	(*----- EOAT Cable(s) -------*)
	(*Fault901 - EOAT01 Cable(s) disconnected*)
		Fault_Tmrs[901].PT:=No_Timer;
		Fault_Tmrs[901]();
		Fault_Tmrs[901].IN:= (MAIN.R1.FB_In.Options.EOAT_Amount>=1) AND
							((EOAT01.ECatSlave_Cable_Breaks[0]<>0)
								OR (EOAT01.ECatSlave_Cable_Breaks[1]<>0));
		Out_To_ICxx.System_Faults[901]:=Fault_Tmrs[901].Q;
	(*Fault902 - EOAT02 Cable(s) disconnected*)
		Fault_Tmrs[902].PT:=No_Timer;
		Fault_Tmrs[902]();
		Fault_Tmrs[902].IN:= (MAIN.R2.FB_In.Options.EOAT_Amount>=2) AND
							((EOAT02.ECatSlave_Cable_Breaks[0]<>0)
								OR (EOAT02.ECatSlave_Cable_Breaks[1]<>0));
		Out_To_ICxx.System_Faults[902]:=Fault_Tmrs[902].Q;
	(*Fault903 - EOAT03 Cable(s) disconnected*)
		Fault_Tmrs[903].PT:=No_Timer;
		Fault_Tmrs[903]();
		Fault_Tmrs[903].IN:= (MAIN.R3.FB_In.Options.EOAT_Amount>=3) AND
							((EOAT04.ECatSlave_Cable_Breaks[0]<>0)
								OR (EOAT04.ECatSlave_Cable_Breaks[1]<>0));
		Out_To_ICxx.System_Faults[903]:=Fault_Tmrs[903].Q;
	(*Fault904 - EOAT04 Cable(s) disconnected*)
		Fault_Tmrs[904].PT:=No_Timer;
		Fault_Tmrs[904]();
		Fault_Tmrs[904].IN:= (MAIN.R4.FB_In.Options.EOAT_Amount>=4) AND
							((EOAT05.ECatSlave_Cable_Breaks[0]<>0)
								OR (EOAT05.ECatSlave_Cable_Breaks[1]<>0));
		Out_To_ICxx.System_Faults[904]:=Fault_Tmrs[904].Q;
	(*Fault905 - EOAT05 Cable(s) disconnected*)
		Fault_Tmrs[905].PT:=No_Timer;
		Fault_Tmrs[905]();
		Fault_Tmrs[905].IN:= (MAIN.R5.FB_In.Options.EOAT_Amount>=5) AND
							((EOAT05.ECatSlave_Cable_Breaks[0]<>0)
								OR (EOAT05.ECatSlave_Cable_Breaks[1]<>0));
		Out_To_ICxx.System_Faults[905]:=Fault_Tmrs[905].Q;
	(*Fault906 - EOAT06 Cable(s) disconnected*)
		Fault_Tmrs[906].PT:=No_Timer;
		Fault_Tmrs[906]();
		Fault_Tmrs[906].IN:= (MAIN.R6.FB_In.Options.EOAT_Amount>=6) AND
							((EOAT06.ECatSlave_Cable_Breaks[0]<>0)
								OR (EOAT06.ECatSlave_Cable_Breaks[1]<>0));
		Out_To_ICxx.System_Faults[906]:=Fault_Tmrs[906].Q;
	(*Fault907 - EOAT07 Cable(s) disconnected*)
		Fault_Tmrs[907].PT:=No_Timer;
		Fault_Tmrs[907]();
		Fault_Tmrs[907].IN:= (MAIN.R7.FB_In.Options.EOAT_Amount>=7) AND
							((EOAT07.ECatSlave_Cable_Breaks[0]<>0)
								OR (EOAT07.ECatSlave_Cable_Breaks[1]<>0));
		Out_To_ICxx.System_Faults[907]:=Fault_Tmrs[907].Q;
	(*Fault908 - EOAT08 Cable(s) disconnected*)
		Fault_Tmrs[908].PT:=No_Timer;
		Fault_Tmrs[908]();
		Fault_Tmrs[908].IN:= (MAIN.R8.FB_In.Options.EOAT_Amount>=8) AND
							((EOAT08.ECatSlave_Cable_Breaks[0]<>0)
								OR (EOAT08.ECatSlave_Cable_Breaks[1]<>0));
		Out_To_ICxx.System_Faults[908]:=Fault_Tmrs[908].Q;
	(*Fault909 - EOAT09 Cable(s) disconnected*)
		Fault_Tmrs[909].PT:=No_Timer;
		Fault_Tmrs[909]();
		Fault_Tmrs[909].IN:= (MAIN.R9.FB_In.Options.EOAT_Amount>=9) AND
							((EOAT09.ECatSlave_Cable_Breaks[0]<>0)
								OR (EOAT09.ECatSlave_Cable_Breaks[1]<>0));
		Out_To_ICxx.System_Faults[909]:=Fault_Tmrs[909].Q;
	(*Fault910 - EOAT10 Cable(s) disconnected*)
		Fault_Tmrs[820].PT:=No_Timer;
		Fault_Tmrs[820]();
		Fault_Tmrs[820].IN:=(MAIN.R10.FB_In.Options.EOAT_Amount>=10) AND
							((EOAT10.ECatSlave_Cable_Breaks[0]<>0)
								OR (EOAT10.ECatSlave_Cable_Breaks[1]<>0));
		Out_To_ICxx.System_Faults[820]:=Fault_Tmrs[820].Q; 
	(*Fault911 - EOAT11 Cable(s) disconnected*)
		Fault_Tmrs[911].PT:=No_Timer;
		Fault_Tmrs[911]();
		Fault_Tmrs[911].IN:= FALSE;
		Out_To_ICxx.System_Faults[911]:=Fault_Tmrs[911].Q;
	(*Fault912 - EOAT12 Cable(s) disconnected*)
		Fault_Tmrs[912].PT:=No_Timer;
		Fault_Tmrs[912]();
		Fault_Tmrs[912].IN:= FALSE;
		Out_To_ICxx.System_Faults[912]:=Fault_Tmrs[912].Q;
	(*Fault913 - EOAT13 Cable(s) disconnected*)
		Fault_Tmrs[913].PT:=No_Timer;
		Fault_Tmrs[913]();
		Fault_Tmrs[913].IN:= FALSE;
		Out_To_ICxx.System_Faults[913]:=Fault_Tmrs[913].Q;
	(*Fault914 - EOAT14 Cable(s) disconnected*)
		Fault_Tmrs[914].PT:=No_Timer;
		Fault_Tmrs[914]();
		Fault_Tmrs[914].IN:= FALSE;
		Out_To_ICxx.System_Faults[914]:=Fault_Tmrs[914].Q;
	(*Fault915 - EOAT15 Cable(s) disconnected*)
		Fault_Tmrs[915].PT:=No_Timer;
		Fault_Tmrs[915]();
		Fault_Tmrs[915].IN:= FALSE;
		Out_To_ICxx.System_Faults[915]:=Fault_Tmrs[915].Q;
	(*Fault916 - EOAT16 Cable(s) disconnected*)
		Fault_Tmrs[916].PT:=No_Timer;
		Fault_Tmrs[916]();
		Fault_Tmrs[916].IN:= FALSE;
		Out_To_ICxx.System_Faults[916]:=Fault_Tmrs[916].Q;
	(*Fault917 - EOAT17 Cable(s) disconnected*)
		Fault_Tmrs[917].PT:=No_Timer;
		Fault_Tmrs[917]();
		Fault_Tmrs[917].IN:= FALSE;
		Out_To_ICxx.System_Faults[917]:=Fault_Tmrs[917].Q;
	(*Fault918 - EOAT18 Cable(s) disconnected*)
		Fault_Tmrs[918].PT:=No_Timer;
		Fault_Tmrs[918]();
		Fault_Tmrs[918].IN:= FALSE;
		Out_To_ICxx.System_Faults[918]:=Fault_Tmrs[918].Q;
	(*Fault919 - EOAT19 Cable(s) disconnected*)
		Fault_Tmrs[919].PT:=No_Timer;
		Fault_Tmrs[919]();
		Fault_Tmrs[919].IN:= FALSE;
		Out_To_ICxx.System_Faults[919]:=Fault_Tmrs[919].Q;
	(*Fault920 - EOAT20 Cable(s) disconnected*)
		Fault_Tmrs[920].PT:=No_Timer;
		Fault_Tmrs[920]();
		Fault_Tmrs[920].IN:= FALSE;
		Out_To_ICxx.System_Faults[920]:=Fault_Tmrs[920].Q;
	(*Fault921 - EOAT21 Cable(s) disconnected*)
		Fault_Tmrs[921].PT:=No_Timer;
		Fault_Tmrs[921]();
		Fault_Tmrs[921].IN:= FALSE;
		Out_To_ICxx.System_Faults[921]:=Fault_Tmrs[921].Q;
	(*Fault922 - EOAT22 Cable(s) disconnected*)
		Fault_Tmrs[922].PT:=No_Timer;
		Fault_Tmrs[922]();
		Fault_Tmrs[922].IN:= FALSE;
		Out_To_ICxx.System_Faults[922]:=Fault_Tmrs[922].Q;
	(*Fault923 - EOAT23 Cable(s) disconnected*)
		Fault_Tmrs[923].PT:=No_Timer;
		Fault_Tmrs[923]();
		Fault_Tmrs[923].IN:= FALSE;
		Out_To_ICxx.System_Faults[923]:=Fault_Tmrs[923].Q;
	(*Fault924 - EOAT24 Cable(s) disconnected*)
		Fault_Tmrs[924].PT:=No_Timer;
		Fault_Tmrs[924]();
		Fault_Tmrs[924].IN:= FALSE;
		Out_To_ICxx.System_Faults[924]:=Fault_Tmrs[924].Q;
	(*Fault925 - EOAT25 Cable(s) disconnected*)
		Fault_Tmrs[925].PT:=No_Timer;
		Fault_Tmrs[925]();
		Fault_Tmrs[925].IN:= FALSE;
		Out_To_ICxx.System_Faults[925]:=Fault_Tmrs[925].Q;
	(*Fault926 - EOAT26 Cable(s) disconnected*)
		Fault_Tmrs[926].PT:=No_Timer;
		Fault_Tmrs[926]();
		Fault_Tmrs[926].IN:= FALSE;
		Out_To_ICxx.System_Faults[926]:=Fault_Tmrs[926].Q;
	(*Fault927 - EOAT27 Cable(s) disconnected*)
		Fault_Tmrs[927].PT:=No_Timer;
		Fault_Tmrs[927]();
		Fault_Tmrs[927].IN:= FALSE;
		Out_To_ICxx.System_Faults[927]:=Fault_Tmrs[927].Q;
	(*Fault928 - EOAT28 Cable(s) disconnected*)
		Fault_Tmrs[928].PT:=No_Timer;
		Fault_Tmrs[928]();
		Fault_Tmrs[928].IN:= FALSE;
		Out_To_ICxx.System_Faults[928]:=Fault_Tmrs[928].Q;
	(*Fault929 - EOAT29 Cable(s) disconnected*)
		Fault_Tmrs[929].PT:=No_Timer;
		Fault_Tmrs[929]();
		Fault_Tmrs[929].IN:= FALSE;
		Out_To_ICxx.System_Faults[929]:=Fault_Tmrs[929].Q;
	(*Fault930 - EOAT30 Cable(s) disconnected*)
		Fault_Tmrs[930].PT:=No_Timer;
		Fault_Tmrs[930]();
		Fault_Tmrs[930].IN:= FALSE;
		Out_To_ICxx.System_Faults[930]:=Fault_Tmrs[930].Q;


	(* --------------------------Services Stand Cable Faults----------------------------*)
	(*Fault931 - SS01 IN Cable Fault*)
		Fault_Tmrs[931].PT:=No_Timer;
		Fault_Tmrs[931]();
		Fault_Tmrs[931].IN:= GTAC_CONFIG.Option_Air1  AND
							MAIN.SS01.EP2028_NotPresent;
		Out_To_ICxx.System_Faults[931]:=Fault_Tmrs[931].Q;
	(*Fault932 - SS01 OUT Cable Fault*)
		Fault_Tmrs[932].PT:=No_Timer;
		Fault_Tmrs[932]();
		Fault_Tmrs[932].IN:= GTAC_CONFIG.Option_Air1  AND
							MAIN.SS01.EP1008_PortB_MissingLink;
		Out_To_ICxx.System_Faults[932]:=Fault_Tmrs[932].Q;
	(*Fault933 - SS02 IN Cable Fault*)
		Fault_Tmrs[933].PT:=No_Timer;
		Fault_Tmrs[933]();
		Fault_Tmrs[933].IN:= GTAC_CONFIG.Option_Air2  AND
							MAIN.SS02.EP2028_NotPresent;
		Out_To_ICxx.System_Faults[933]:=Fault_Tmrs[933].Q;
	(*Fault934 - SS02 OUT Cable Fault*)
		Fault_Tmrs[934].PT:=No_Timer;
		Fault_Tmrs[934]();
		Fault_Tmrs[934].IN:= GTAC_CONFIG.Option_Air2  AND
							MAIN.SS02.EP1008_PortB_MissingLink;
		Out_To_ICxx.System_Faults[934]:=Fault_Tmrs[934].Q;
(*
	(*Fault935 - SS03 IN Cable Fault*)
		Fault_Tmrs[935].PT:=No_Timer;
		Fault_Tmrs[935]();
		Fault_Tmrs[935].IN:= (GTAC_CONFIG.Option_Air1>=1)  AND
							MAIN.SS03.EP2028_NotPresent;
		Out_To_ICxx.System_Faults[935]:=Fault_Tmrs[935].Q;
	(*Fault936 - SS03 OUT Cable Fault*)
		Fault_Tmrs[936].PT:=No_Timer;
		Fault_Tmrs[936]();
		Fault_Tmrs[936].IN:= (GTAC_CONFIG.Option_Air1>=1)  AND
							MAIN.SS03.EP1008_PortB_MissingLink;
		Out_To_ICxx.System_Faults[936]:=Fault_Tmrs[546].Q;
*)
	(* --------------------------Enable Switch Plate Cable Faults----------------------------*)
	(*Fault937 - ESW01 IN Cable Fault*)
		Fault_Tmrs[937].PT:=No_Timer;
		Fault_Tmrs[937]();
		Fault_Tmrs[937].IN:= (GTAC_CONFIG.Option_ESW_Count>=1)  AND
							MAIN.ESW01.EP1908_NotPresent;
		Out_To_ICxx.System_Faults[937]:=Fault_Tmrs[937].Q;
	(*Fault938 - ESW01 OUT Cable Fault*)
		Fault_Tmrs[938].PT:=No_Timer;
		Fault_Tmrs[938]();
		Fault_Tmrs[938].IN:= (GTAC_CONFIG.Option_ESW_Count>=1)  AND
							MAIN.ESW01.EP1908_PortB_MissingLink;
		Out_To_ICxx.System_Faults[938]:=Fault_Tmrs[938].Q;
	(*Fault939 - ESW02 IN Cable Fault*)
		Fault_Tmrs[939].PT:=No_Timer;
		Fault_Tmrs[939]();
		Fault_Tmrs[939].IN:= (GTAC_CONFIG.Option_ESW_Count>=2)  AND
							MAIN.ESW02.EP1908_NotPresent;
		Out_To_ICxx.System_Faults[939]:=Fault_Tmrs[939].Q;
	(*Fault940 - ESW02 OUT Cable Fault*)
		Fault_Tmrs[940].PT:=No_Timer;
		Fault_Tmrs[940]();
		Fault_Tmrs[940].IN:= (GTAC_CONFIG.Option_ESW_Count>=2)  AND
							MAIN.ESW02.EP1908_PortB_MissingLink;
		Out_To_ICxx.System_Faults[940]:=Fault_Tmrs[940].Q;
	(*Fault941 - ESW03 IN Cable Fault*)
		Fault_Tmrs[941].PT:=No_Timer;
		Fault_Tmrs[941]();
		Fault_Tmrs[941].IN:= (GTAC_CONFIG.Option_ESW_Count>=3)  AND
							MAIN.ESW03.EP1908_NotPresent;
		Out_To_ICxx.System_Faults[941]:=Fault_Tmrs[941].Q;
	(*Fault942 - ESW03 OUT Cable Fault*)
		Fault_Tmrs[942].PT:=No_Timer;
		Fault_Tmrs[942]();
		Fault_Tmrs[942].IN:= (GTAC_CONFIG.Option_ESW_Count>=3)  AND
							MAIN.ESW03.EP1908_PortB_MissingLink;
		Out_To_ICxx.System_Faults[942]:=Fault_Tmrs[942].Q;
	(*Fault943 - ESW04 IN Cable Fault*)
		Fault_Tmrs[943].PT:=No_Timer;
		Fault_Tmrs[943]();
		Fault_Tmrs[943].IN:= (GTAC_CONFIG.Option_ESW_Count>=4)  AND
							MAIN.ESW04.EP1908_NotPresent;
		Out_To_ICxx.System_Faults[943]:=Fault_Tmrs[943].Q;
	(*Fault944 - ESW04 OUT Cable Fault*)
		Fault_Tmrs[944].PT:=No_Timer;
		Fault_Tmrs[944]();
		Fault_Tmrs[944].IN:= (GTAC_CONFIG.Option_ESW_Count>=4)  AND
							MAIN.ESW04.EP1908_PortB_MissingLink;
		Out_To_ICxx.System_Faults[944]:=Fault_Tmrs[944].Q;

(* -------------------------- IS Cable Faults----------------------------*)

	(*Fault751 - IS01 Cable break fault (any cable break)*)
		Fault_Tmrs[945].PT:= No_Timer;
		Fault_Tmrs[945]();
		Fault_Tmrs[945].IN:= (GTAC_CONFIG.Option_IS_Count >= 1) AND 
							(MAIN.IS01.ECatSlave_Cable_Breaks <> 0);
		Out_To_ICxx.System_Faults[945]:=Fault_Tmrs[945].Q;
	(*Fault752 - IS01 Profibus Network Fault*)
		Fault_Tmrs[946].PT:= No_Timer;
		Fault_Tmrs[946]();
		Fault_Tmrs[946].IN:= (GTAC_CONFIG.Option_IS_Count >= 1) AND 
							MAIN.IS01.FB_In.Option_Enable_Pbus AND
							NOT (MAIN.IS01.ProfiNode_OK);
		Out_To_ICxx.System_Faults[946]:=Fault_Tmrs[946].Q;

	(* -------------------------- Servo Drive Cable Faults----------------------------*)

	(*Fault951 - SD1 Cable(s) disconnected*)
		Fault_Tmrs[951].PT:= No_Timer;
		Fault_Tmrs[951]();
		Fault_Tmrs[951].IN:= (GTAC_CONFIG.Option_SD_Count>=1) AND
							(Servo_Motion.SD[1].ECatSlave_Cable_Breaks<>0);
		Out_To_ICxx.System_Faults[951]:=Fault_Tmrs[951].Q;
	(*Fault952 - SD2 Cable(s) disconnected*)
		Fault_Tmrs[952].PT:= No_Timer;
		Fault_Tmrs[952]();
		Fault_Tmrs[952].IN:= (GTAC_CONFIG.Option_SD_Count>=2) AND
							(Servo_Motion.SD[2].ECatSlave_Cable_Breaks<>0);
		Out_To_ICxx.System_Faults[952]:=Fault_Tmrs[952].Q;
	(*Fault953 - SD3 Cable(s) disconnected*)
		Fault_Tmrs[953].PT:= No_Timer;
		Fault_Tmrs[953]();
		Fault_Tmrs[953].IN:= (GTAC_CONFIG.Option_SD_Count>=3) AND
							(Servo_Motion.SD[3].ECatSlave_Cable_Breaks<>0);
		Out_To_ICxx.System_Faults[953]:=Fault_Tmrs[953].Q;
	(*Fault954 - SD4 Cable(s) disconnected*)
		Fault_Tmrs[954].PT:= No_Timer;
		Fault_Tmrs[954]();
		Fault_Tmrs[954].IN:= (GTAC_CONFIG.Option_SD_Count>=4) AND
							(Servo_Motion.SD[4].ECatSlave_Cable_Breaks<>0);
		Out_To_ICxx.System_Faults[954]:=Fault_Tmrs[954].Q;
	(*Fault955 - SD5 Cable(s) disconnected*)
		Fault_Tmrs[955].PT:= No_Timer;
		Fault_Tmrs[955]();
		Fault_Tmrs[955].IN:= (GTAC_CONFIG.Option_SD_Count>=5) AND
							(Servo_Motion.SD[5].ECatSlave_Cable_Breaks<>0);
		Out_To_ICxx.System_Faults[955]:=Fault_Tmrs[955].Q;
	(*Fault956 - SD6 Cable(s) disconnected*)
		Fault_Tmrs[956].PT:= No_Timer;
		Fault_Tmrs[956]();
		Fault_Tmrs[956].IN:= (GTAC_CONFIG.Option_SD_Count>=6) AND
							(Servo_Motion.SD[6].ECatSlave_Cable_Breaks<>0);
		Out_To_ICxx.System_Faults[956]:=Fault_Tmrs[956].Q;
	(*Fault957 - SD7 Cable(s) disconnected*)
		Fault_Tmrs[957].PT:= No_Timer;
		Fault_Tmrs[957]();
		Fault_Tmrs[957].IN:= (GTAC_CONFIG.Option_SD_Count>=7) AND
							(Servo_Motion.SD[7].ECatSlave_Cable_Breaks<>0);
		Out_To_ICxx.System_Faults[957]:=Fault_Tmrs[957].Q;
	(*Fault958 - SD8 Cable(s) disconnected*)
		Fault_Tmrs[958].PT:= No_Timer;
		Fault_Tmrs[958]();
		Fault_Tmrs[958].IN:= (GTAC_CONFIG.Option_SD_Count>=8) AND
							(Servo_Motion.SD[8].ECatSlave_Cable_Breaks<>0);
		Out_To_ICxx.System_Faults[958]:=Fault_Tmrs[958].Q;
	(*Fault959 - SD9 Cable(s) disconnected*)
		Fault_Tmrs[959].PT:= No_Timer;
		Fault_Tmrs[959]();
		Fault_Tmrs[959].IN:= (GTAC_CONFIG.Option_SD_Count>=9) AND
							(Servo_Motion.SD[9].ECatSlave_Cable_Breaks<>0);
		Out_To_ICxx.System_Faults[959]:=Fault_Tmrs[959].Q;
	(*Fault960 - SD10 Cable(s) disconnected*)
		Fault_Tmrs[960].PT:= No_Timer;
		Fault_Tmrs[960]();
		Fault_Tmrs[960].IN:= (GTAC_CONFIG.Option_SD_Count>=10) AND
							(Servo_Motion.SD[10].ECatSlave_Cable_Breaks<>0);
		Out_To_ICxx.System_Faults[960]:=Fault_Tmrs[960].Q;
	(*Fault961 - SD11 Cable(s) disconnected*)
		Fault_Tmrs[961].PT:= No_Timer;
		Fault_Tmrs[961]();
		Fault_Tmrs[961].IN:= (GTAC_CONFIG.Option_SD_Count>=11) AND
							(Servo_Motion.SD[11].ECatSlave_Cable_Breaks<>0);
		Out_To_ICxx.System_Faults[961]:=Fault_Tmrs[961].Q;
	(*Fault962 - SD12 Cable(s) disconnected*)
		Fault_Tmrs[962].PT:= No_Timer;
		Fault_Tmrs[962]();
		Fault_Tmrs[962].IN:= (GTAC_CONFIG.Option_SD_Count>=12) AND
							(Servo_Motion.SD[12].ECatSlave_Cable_Breaks<>0);
		Out_To_ICxx.System_Faults[962]:=Fault_Tmrs[962].Q;
	(*Fault963 - SD13 Cable(s) disconnected*)
		Fault_Tmrs[963].PT:= No_Timer;
		Fault_Tmrs[963]();
		Fault_Tmrs[963].IN:= (GTAC_CONFIG.Option_SD_Count>=13) AND
							(Servo_Motion.SD[13].ECatSlave_Cable_Breaks<>0);
		Out_To_ICxx.System_Faults[963]:=Fault_Tmrs[963].Q;
	(*Fault964 - SD14 Cable(s) disconnected*)
		Fault_Tmrs[964].PT:= No_Timer;
		Fault_Tmrs[964]();
		Fault_Tmrs[964].IN:= (GTAC_CONFIG.Option_SD_Count>=14) AND
							(Servo_Motion.SD[14].ECatSlave_Cable_Breaks<>0);
		Out_To_ICxx.System_Faults[964]:=Fault_Tmrs[964].Q;
	(*Fault965 - SD15 Cable(s) disconnected*)
		Fault_Tmrs[965].PT:= No_Timer;
		Fault_Tmrs[965]();
		Fault_Tmrs[965].IN:= (GTAC_CONFIG.Option_SD_Count>=15) AND
							(Servo_Motion.SD[15].ECatSlave_Cable_Breaks<>0);
		Out_To_ICxx.System_Faults[965]:=Fault_Tmrs[965].Q;
	(*Fault966 - SD16 Cable(s) disconnected*)
		Fault_Tmrs[966].PT:= No_Timer;
		Fault_Tmrs[966]();
		Fault_Tmrs[966].IN:= (GTAC_CONFIG.Option_SD_Count>=16) AND
							(Servo_Motion.SD[16].ECatSlave_Cable_Breaks<>0);
		Out_To_ICxx.System_Faults[966]:=Fault_Tmrs[966].Q;
	(*Fault967 - SD17 Cable(s) disconnected*)
		Fault_Tmrs[967].PT:= No_Timer;
		Fault_Tmrs[967]();
		Fault_Tmrs[967].IN:= (GTAC_CONFIG.Option_SD_Count>=17) AND
							(Servo_Motion.SD[17].ECatSlave_Cable_Breaks<>0);
		Out_To_ICxx.System_Faults[967]:=Fault_Tmrs[967].Q;
	(*Fault968 - SD18 Cable(s) disconnected*)
		Fault_Tmrs[968].PT:= No_Timer;
		Fault_Tmrs[968]();
		Fault_Tmrs[968].IN:= (GTAC_CONFIG.Option_SD_Count>=18) AND
							(Servo_Motion.SD[18].ECatSlave_Cable_Breaks<>0);
		Out_To_ICxx.System_Faults[968]:=Fault_Tmrs[968].Q;
	(*Fault969 - SD19 Cable(s) disconnected*)
		Fault_Tmrs[969].PT:= No_Timer;
		Fault_Tmrs[969]();
		Fault_Tmrs[969].IN:= (GTAC_CONFIG.Option_SD_Count>=19) AND
							(Servo_Motion.SD[19].ECatSlave_Cable_Breaks<>0);
		Out_To_ICxx.System_Faults[969]:=Fault_Tmrs[969].Q;
	(*Fault970 - SD20 Cable(s) disconnected*)
		Fault_Tmrs[970].PT:= No_Timer;
		Fault_Tmrs[970]();
		Fault_Tmrs[970].IN:= (GTAC_CONFIG.Option_SD_Count>=20) AND
							(Servo_Motion.SD[20].ECatSlave_Cable_Breaks<>0);
		Out_To_ICxx.System_Faults[970]:=Fault_Tmrs[970].Q;
	(*Fault971 - SD21 Cable(s) disconnected*)
		Fault_Tmrs[971].PT:= No_Timer;
		Fault_Tmrs[971]();
		Fault_Tmrs[971].IN:= (GTAC_CONFIG.Option_SD_Count>=21) AND
							(Servo_Motion.SD[21].ECatSlave_Cable_Breaks<>0);
		Out_To_ICxx.System_Faults[971]:=Fault_Tmrs[971].Q;
	(*Fault972 - SD22 Cable(s) disconnected*)
		Fault_Tmrs[972].PT:= No_Timer;
		Fault_Tmrs[972]();
		Fault_Tmrs[972].IN:= (GTAC_CONFIG.Option_SD_Count>=22) AND
							(Servo_Motion.SD[22].ECatSlave_Cable_Breaks<>0);
		Out_To_ICxx.System_Faults[972]:=Fault_Tmrs[972].Q;
	(*Fault973 - SD23 Cable(s) disconnected*)
		Fault_Tmrs[973].PT:= No_Timer;
		Fault_Tmrs[973]();
		Fault_Tmrs[973].IN:= (GTAC_CONFIG.Option_SD_Count>=23) AND
							(Servo_Motion.SD[23].ECatSlave_Cable_Breaks<>0);
		Out_To_ICxx.System_Faults[973]:=Fault_Tmrs[973].Q;
	(*Fault974 - SD24 Cable(s) disconnected*)
		Fault_Tmrs[974].PT:= No_Timer;
		Fault_Tmrs[974]();
		Fault_Tmrs[974].IN:= (GTAC_CONFIG.Option_SD_Count>=24) AND
							(Servo_Motion.SD[24].ECatSlave_Cable_Breaks<>0);
		Out_To_ICxx.System_Faults[974]:=Fault_Tmrs[974].Q;
	(*Fault975 - SD25 Cable(s) disconnected*)
		Fault_Tmrs[975].PT:= No_Timer;
		Fault_Tmrs[975]();
		Fault_Tmrs[975].IN:= (GTAC_CONFIG.Option_SD_Count>=25) AND
							(Servo_Motion.SD[25].ECatSlave_Cable_Breaks<>0);
		Out_To_ICxx.System_Faults[975]:=Fault_Tmrs[975].Q;
	(*Fault976 - SD26 Cable(s) disconnected*)
		Fault_Tmrs[976].PT:= No_Timer;
		Fault_Tmrs[976]();
		Fault_Tmrs[976].IN:= (GTAC_CONFIG.Option_SD_Count>=26) AND
							(Servo_Motion.SD[26].ECatSlave_Cable_Breaks<>0);
		Out_To_ICxx.System_Faults[976]:=Fault_Tmrs[976].Q;
	(*Fault977 - SD27 Cable(s) disconnected*)
		Fault_Tmrs[977].PT:= No_Timer;
		Fault_Tmrs[977]();
		Fault_Tmrs[977].IN:= (GTAC_CONFIG.Option_SD_Count>=27) AND
							(Servo_Motion.SD[27].ECatSlave_Cable_Breaks<>0);
		Out_To_ICxx.System_Faults[977]:=Fault_Tmrs[977].Q;
	(*Fault978 - SD28 Cable(s) disconnected*)
		Fault_Tmrs[978].PT:= No_Timer;
		Fault_Tmrs[978]();
		Fault_Tmrs[978].IN:= (GTAC_CONFIG.Option_SD_Count>=28) AND
							(Servo_Motion.SD[28].ECatSlave_Cable_Breaks<>0);
		Out_To_ICxx.System_Faults[978]:=Fault_Tmrs[978].Q;
	(*Fault979 - SD29 Cable(s) disconnected*)
		Fault_Tmrs[979].PT:= No_Timer;
		Fault_Tmrs[979]();
		Fault_Tmrs[979].IN:= (GTAC_CONFIG.Option_SD_Count>=29) AND
							(Servo_Motion.SD[29].ECatSlave_Cable_Breaks<>0);
		Out_To_ICxx.System_Faults[979]:=Fault_Tmrs[979].Q;
	(*Fault980 - SD30 Cable(s) disconnected*)
		Fault_Tmrs[980].PT:= No_Timer;
		Fault_Tmrs[980]();
		Fault_Tmrs[980].IN:= (GTAC_CONFIG.Option_SD_Count>=30) AND
							(Servo_Motion.SD[30].ECatSlave_Cable_Breaks<>0);
		Out_To_ICxx.System_Faults[980]:=Fault_Tmrs[980].Q;


	(* --------------------------Laser Controller Cable Faults----------------------------*)
	(*Fault981 - LSR01 IN Cable Fault*)
		Fault_Tmrs[981].PT:=No_Timer;
		Fault_Tmrs[981]();
		Fault_Tmrs[981].IN:= (GTAC_CONFIG.Option_LaserController_Count>=1)  AND
							MAIN.Laser01.EL6692_NotPresent;
		Out_To_ICxx.System_Faults[981]:=Fault_Tmrs[981].Q;
	(*Fault982 - LSR01 OUT Cable Fault*)
		Fault_Tmrs[982].PT:=No_Timer;
		Fault_Tmrs[982]();
		Fault_Tmrs[982].IN:= (GTAC_CONFIG.Option_LaserController_Count>=1)  AND
							MAIN.Laser01.EL6692_PortC_MissingLink;
		Out_To_ICxx.System_Faults[982]:=Fault_Tmrs[982].Q;

	(*------------------------------------------------------------- Start Of Faults that Will NOT Stop All Automation --------------------------------------------------*)
	(*--------------------------------------------------------- Start of  ICxx Operator Station Faults ---------------------------------------------------------*)
	(*------------------- IC01 -----------------*)
	(*Fault991 - IC01OP1 Motion Faults*)
		Fault_Tmrs[991].PT:=Short_Faults;
		Fault_Tmrs[991]();
		Fault_Tmrs[991].IN:= GTAC_CONFIG.Option_HumanFix_Enables.1 AND
							Out_To_ICxx.Fix01_Discrete_Image.CLFaulted.0;
		Out_To_ICxx.System_Faults[991]:=Fault_Tmrs[991].Q;
	(*Fault992 - IC01OP1 Part Present Faults*)
		Fault_Tmrs[992].PT:=Short_Faults;
		Fault_Tmrs[992]();
		Fault_Tmrs[992].IN:= GTAC_CONFIG.Option_HumanFix_Enables.1 AND
							Out_To_ICxx.Fix01_Discrete_Image.PPFaulted.0;
		Out_To_ICxx.System_Faults[992]:=Fault_Tmrs[992].Q;
	(*Fault993 - IC01OP1 Vertical LC Broken While Robot(s) In Zone*)
		VLC_Capture11_TOF.PT:= T#2.0S;
		VLC_Capture11_TOF();
		(*Differentiate between Turtable type Fix01/02 and standard Fix01*)
		(*Turntable Type*)
		IF (MAIN.R1.FB_In.Robot_Type = KUKA_KRC4_SAFEOP_TurnTable) THEN
		VLC_Capture11_TOF.IN:= (GTAC_CONFIG.Option_IC_Count>=1) AND GTAC_CONFIG.Option_HumanFix_Enables.1 AND
								NOT MAIN.IC01.OP1_HumanVertLC_Clear AND NOT Fix01.All_Robots_Clear
								AND (Fix01.Turntable_WorkingOK OR Fix02.Turntable_WorkingOK);
		(*Standard Type*)						
		ELSE
		VLC_Capture11_TOF.IN:= (GTAC_CONFIG.Option_IC_Count>=1) AND GTAC_CONFIG.Option_HumanFix_Enables.1 AND
								NOT MAIN.IC01.OP1_HumanVertLC_Clear AND NOT Fix01.All_Robots_Clear;
		END_IF
		Out_To_ICxx.System_Faults[993]:= VLC_Capture11_TOF.Q;
	(*Fault994 - IC01OP1 Horizontal LC Broken While Robot(s) In Zone*)
		HLC_Capture12_TOF.PT:= T#2.0S;
		HLC_Capture12_TOF();
		(*Differentiate between Turtable type Fix01/02 and standard Fix01*)
		(*Turntable Type*)
		IF (MAIN.R1.FB_In.Robot_Type = KUKA_KRC4_SAFEOP_TurnTable) THEN
		HLC_Capture12_TOF.IN:= (GTAC_CONFIG.Option_IC_Count>=1) AND GTAC_CONFIG.Option_HumanFix_Enables.1 AND
								NOT MAIN.IC01.OP1_HumanHorizLC_Clear AND NOT Fix01.All_Robots_Clear
								AND (Fix01.Turntable_WorkingOK OR Fix02.Turntable_WorkingOK);
		(*Standard Type*)						
		ELSE
		HLC_Capture12_TOF.IN:= (GTAC_CONFIG.Option_IC_Count>=1) AND GTAC_CONFIG.Option_HumanFix_Enables.1 AND
								NOT MAIN.IC01.OP1_HumanHorizLC_Clear AND NOT Fix01.All_Robots_Clear;
		END_IF
		Out_To_ICxx.System_Faults[994]:= HLC_Capture12_TOF.Q;
	(*Fault995 - IC01OP1 Horizontal LC3 Broken While Robot(s) In Zone*)
		HLC_Capture13_TOF.PT:= T#2.0S;
		HLC_Capture13_TOF();
		(*Differentiate between Turtable type Fix01/02 and standard Fix01*)
		(*Turntable Type*)
		IF (MAIN.R1.FB_In.Robot_Type = KUKA_KRC4_SAFEOP_TurnTable) THEN
		HLC_Capture13_TOF.IN:= (GTAC_CONFIG.Option_IC_Count>=1) AND GTAC_CONFIG.Option_HumanFix_Enables.1 AND
								NOT MAIN.IC01.OP1_RobotVertLC_Clear AND NOT Fix01.All_Robots_Clear
								AND (Fix01.Turntable_WorkingOK OR Fix02.Turntable_WorkingOK);
		(*Standard Type*)						
		ELSE
		HLC_Capture13_TOF.IN:= (GTAC_CONFIG.Option_IC_Count>=1) AND GTAC_CONFIG.Option_HumanFix_Enables.1 AND
								NOT MAIN.IC01.OP1_RobotVertLC_Clear AND NOT Fix01.All_Robots_Clear;
		END_IF
		Out_To_ICxx.System_Faults[995]:= HLC_Capture13_TOF.Q;

	(*Fault996 - IC01OP2 Motion Faults*)
		Fault_Tmrs[996].PT:=Short_Faults;
		Fault_Tmrs[996]();
		Fault_Tmrs[996].IN:= GTAC_CONFIG.Option_HumanFix_Enables.2 AND
							Out_To_ICxx.Fix02_Discrete_Image.CLFaulted.0;
		Out_To_ICxx.System_Faults[996]:=Fault_Tmrs[996].Q;
	(*Fault997 - IC01OP2 Part Present Faults*)
		Fault_Tmrs[997].PT:=Short_Faults;
		Fault_Tmrs[997]();
		Fault_Tmrs[997].IN:= GTAC_CONFIG.Option_HumanFix_Enables.2 AND
							Out_To_ICxx.Fix02_Discrete_Image.PPFaulted.0;
		Out_To_ICxx.System_Faults[997]:=Fault_Tmrs[997].Q;
	(*Fault998 - IC01OP2 Vertical LC Broken While Robot(s) In Zone*)
		VLC_Capture21_TOF.PT:= T#2.0S;
		VLC_Capture21_TOF();
		(*Differentiate between Turtable type Fix01/02 and standard Fix01*)
		(*Turntable Type*)
		IF (MAIN.R1.FB_In.Robot_Type = KUKA_KRC4_SAFEOP_TurnTable) THEN
		VLC_Capture21_TOF.IN:= (GTAC_CONFIG.Option_IC_Count>=1) AND GTAC_CONFIG.Option_HumanFix_Enables.2 AND
								NOT MAIN.IC01.OP2_HumanVertLC_Clear AND NOT Fix02.All_Robots_Clear
								AND (Fix01.Turntable_WorkingOK OR Fix02.Turntable_WorkingOK);
		(*Standard Type*)						
		ELSE
		VLC_Capture21_TOF.IN:= (GTAC_CONFIG.Option_IC_Count>=1) AND GTAC_CONFIG.Option_HumanFix_Enables.2 AND
								NOT MAIN.IC01.OP2_HumanVertLC_Clear AND NOT Fix02.All_Robots_Clear;
		END_IF
		Out_To_ICxx.System_Faults[998]:= VLC_Capture21_TOF.Q;
	(*Fault999 - IC01OP2 Horizontal LC Broken While Robot(s) In Zone*)
		HLC_Capture22_TOF.PT:= T#2.0S;
		HLC_Capture22_TOF();
		(*Differentiate between Turtable type Fix01/02 and standard Fix01*)
		(*Turntable Type*)
		IF (MAIN.R1.FB_In.Robot_Type = KUKA_KRC4_SAFEOP_TurnTable) THEN
		HLC_Capture22_TOF.IN:= (GTAC_CONFIG.Option_IC_Count>=1) AND GTAC_CONFIG.Option_HumanFix_Enables.2 AND
								NOT MAIN.IC01.OP2_HumanHorizLC_Clear AND NOT Fix02.All_Robots_Clear
								AND (Fix01.Turntable_WorkingOK OR Fix02.Turntable_WorkingOK);
		(*Standard Type*)						
		ELSE
		HLC_Capture22_TOF.IN:= (GTAC_CONFIG.Option_IC_Count>=1) AND GTAC_CONFIG.Option_HumanFix_Enables.2 AND
								NOT MAIN.IC01.OP2_HumanHorizLC_Clear AND NOT Fix02.All_Robots_Clear;
		END_IF
		Out_To_ICxx.System_Faults[999]:= HLC_Capture22_TOF.Q;
	(*Fault1000 - IC01OP2 Horizontal LC3 Broken While Robot(s) In Zone*)
		HLC_Capture23_TOF.PT:= T#2.0S;
		HLC_Capture23_TOF();
		(*Differentiate between Turtable type Fix01/02 and standard Fix01*)
		(*Turntable Type*)
		IF (MAIN.R1.FB_In.Robot_Type = KUKA_KRC4_SAFEOP_TurnTable) THEN
		HLC_Capture23_TOF.IN:= (GTAC_CONFIG.Option_IC_Count>=1) AND GTAC_CONFIG.Option_HumanFix_Enables.2 AND
								NOT MAIN.IC01.OP2_RobotVertLC_Clear AND NOT Fix02.All_Robots_Clear
								AND (Fix01.Turntable_WorkingOK OR Fix02.Turntable_WorkingOK);
		(*Standard Type*)						
		ELSE
		HLC_Capture23_TOF.IN:= (GTAC_CONFIG.Option_IC_Count>=1) AND GTAC_CONFIG.Option_HumanFix_Enables.2 AND
								NOT MAIN.IC01.OP2_RobotVertLC_Clear AND NOT Fix02.All_Robots_Clear;
		END_IF
		Out_To_ICxx.System_Faults[1000]:= HLC_Capture23_TOF.Q;
		
	(*------------------- IC02 -----------------*)
	(*Fault1001 - IC02OP1 Motion Faults*)
		Fault_Tmrs[1001].PT:=Short_Faults;
		Fault_Tmrs[1001]();
		Fault_Tmrs[1001].IN:= GTAC_CONFIG.Option_HumanFix_Enables.3 AND
							Out_To_ICxx.Fix03_Discrete_Image.CLFaulted.0;
		Out_To_ICxx.System_Faults[1001]:=Fault_Tmrs[1001].Q;
	(*Fault1002 - IC02OP1 Part Present Faults*)
		Fault_Tmrs[1002].PT:=Short_Faults;
		Fault_Tmrs[1002]();
		Fault_Tmrs[1002].IN:= GTAC_CONFIG.Option_HumanFix_Enables.3 AND
							Out_To_ICxx.Fix03_Discrete_Image.PPFaulted.0;
		Out_To_ICxx.System_Faults[1002]:=Fault_Tmrs[1002].Q;
	(*Fault1003 - IC02OP1 Vertical LC Broken While Robot(s) In Zone*)
		VLC_Capture31_TOF.PT:= T#2.0S;
		VLC_Capture31_TOF();
		VLC_Capture31_TOF.IN:= (GTAC_CONFIG.Option_IC_Count>=2) AND GTAC_CONFIG.Option_HumanFix_Enables.3 AND
								NOT MAIN.IC02.OP1_HumanVertLC_Clear AND NOT Fix03.All_Robots_Clear;
		Out_To_ICxx.System_Faults[1003]:= HLC_Capture31_TOF.Q;
	(*Fault1004 - IC02OP1 Horizontal LC Broken While Robot(s) In Zone*)
		HLC_Capture32_TOF.PT:= T#2.0S;
		HLC_Capture32_TOF();
		HLC_Capture32_TOF.IN:= (GTAC_CONFIG.Option_IC_Count>=2) AND GTAC_CONFIG.Option_HumanFix_Enables.3 AND
								NOT MAIN.IC02.OP1_HumanHorizLC_Clear AND NOT Fix03.All_Robots_Clear;
		Out_To_ICxx.System_Faults[1004]:= HLC_Capture32_TOF.Q;
	(*Fault1005 - IC02OP1 Horizontal LC3 Broken While Robot(s) In Zone*)
		HLC_Capture33_TOF.PT:= T#2.0S;
		HLC_Capture33_TOF();
		HLC_Capture33_TOF.IN:= (GTAC_CONFIG.Option_IC_Count>=2) AND GTAC_CONFIG.Option_HumanFix_Enables.3 AND
								NOT MAIN.IC02.OP1_RobotVertLC_Clear AND NOT Fix03.All_Robots_Clear;
		Out_To_ICxx.System_Faults[1005]:= HLC_Capture33_TOF.Q;

	(*Fault1006 - IC02OP2 Motion Faults*)
		Fault_Tmrs[1006].PT:=Short_Faults;
		Fault_Tmrs[1006]();
		Fault_Tmrs[1006].IN:= GTAC_CONFIG.Option_HumanFix_Enables.4 AND
							Out_To_ICxx.Fix04_Discrete_Image.CLFaulted.0;
		Out_To_ICxx.System_Faults[1006]:=Fault_Tmrs[1006].Q;
	(*Fault1007 - IC02OP2 Part Present Faults*)
		Fault_Tmrs[1007].PT:=Short_Faults;
		Fault_Tmrs[1007]();
		Fault_Tmrs[1007].IN:= GTAC_CONFIG.Option_HumanFix_Enables.4 AND
							Out_To_ICxx.Fix04_Discrete_Image.PPFaulted.0;
		Out_To_ICxx.System_Faults[1007]:=Fault_Tmrs[1007].Q;
	(*Fault1008 - IC02OP2 Vertical LC Broken While Robot(s) In Zone*)
		VLC_Capture41_TOF.PT:= T#2.0S;
		VLC_Capture41_TOF();
		VLC_Capture41_TOF.IN:= (GTAC_CONFIG.Option_IC_Count>=2) AND GTAC_CONFIG.Option_HumanFix_Enables.4 AND
								NOT MAIN.IC02.OP2_HumanVertLC_Clear AND NOT Fix04.All_Robots_Clear;
		Out_To_ICxx.System_Faults[1008]:= VLC_Capture41_TOF.Q;
	(*Fault1009 - IC02OP2 Horizontal LC Broken While Robot(s) In Zone*)
		HLC_Capture42_TOF.PT:= T#2.0S;
		HLC_Capture42_TOF();
		HLC_Capture42_TOF.IN:= (GTAC_CONFIG.Option_IC_Count>=2)AND GTAC_CONFIG.Option_HumanFix_Enables.4 AND
								NOT MAIN.IC02.OP2_HumanHorizLC_Clear AND NOT Fix04.All_Robots_Clear;
		Out_To_ICxx.System_Faults[1009]:= HLC_Capture42_TOF.Q;
	(*Fault1010 - IC02OP2 Horizontal LC Broken While Robot(s) In Zone*)
		HLC_Capture43_TOF.PT:= T#2.0S;
		HLC_Capture43_TOF();
		HLC_Capture43_TOF.IN:= (GTAC_CONFIG.Option_IC_Count>=2)AND GTAC_CONFIG.Option_HumanFix_Enables.4 AND
								NOT (*MAIN.IC02.OP2_RobotVertLC_Clear*) MAIN.IC02.OP1_RobotVertLC_Clear AND NOT Fix04.All_Robots_Clear;
		Out_To_ICxx.System_Faults[1010]:= HLC_Capture43_TOF.Q;


	(*------------------- IC03 -----------------*)
	(*Fault1011 - IC03OP1 Motion Faults*)
		Fault_Tmrs[1011].PT:=Short_Faults;
		Fault_Tmrs[1011]();
		Fault_Tmrs[1011].IN:= GTAC_CONFIG.Option_HumanFix_Enables.5 AND
							Out_To_ICxx.Fix05_Discrete_Image.CLFaulted.0;
		Out_To_ICxx.System_Faults[1011]:=Fault_Tmrs[1011].Q;
	(*Fault1012 - IC03OP1 Part Present Faults*)
		Fault_Tmrs[1012].PT:=Short_Faults;
		Fault_Tmrs[1012]();
		Fault_Tmrs[1012].IN:= GTAC_CONFIG.Option_HumanFix_Enables.5 AND
							Out_To_ICxx.Fix05_Discrete_Image.PPFaulted.0;
		Out_To_ICxx.System_Faults[1012]:=Fault_Tmrs[1012].Q;
	(*Fault1013 - IC03OP1 Vertical LC Broken While Robot(s) In Zone*)
		VLC_Capture51_TOF.PT:= T#2.0S;
		VLC_Capture51_TOF();
		VLC_Capture51_TOF.IN:= (GTAC_CONFIG.Option_IC_Count>=3) AND GTAC_CONFIG.Option_HumanFix_Enables.5 AND
								NOT MAIN.IC03.OP1_HumanVertLC_Clear AND NOT Fix05.All_Robots_Clear;
		Out_To_ICxx.System_Faults[1013]:= VLC_Capture51_TOF.Q;
	(*Fault1014 - IC03OP1 Horizontal LC Broken While Robot(s) In Zone*)
		HLC_Capture52_TOF.PT:= T#2.0S;
		HLC_Capture52_TOF();
		HLC_Capture52_TOF.IN:= (GTAC_CONFIG.Option_IC_Count>=3) AND GTAC_CONFIG.Option_HumanFix_Enables.5 AND
								NOT MAIN.IC03.OP1_HumanHorizLC_Clear AND NOT Fix05.All_Robots_Clear;
		Out_To_ICxx.System_Faults[1014]:= HLC_Capture52_TOF.Q;
	(*Fault1015 - IC03OP1 Horizontal LC3 Broken While Robot(s) In Zone*)
		HLC_Capture53_TOF.PT:= T#2.0S;
		HLC_Capture53_TOF();
		HLC_Capture53_TOF.IN:= (GTAC_CONFIG.Option_IC_Count>=3) AND GTAC_CONFIG.Option_HumanFix_Enables.5 AND
								NOT MAIN.IC03.OP1_RobotVertLC_Clear AND NOT Fix05.All_Robots_Clear AND FALSE;
		Out_To_ICxx.System_Faults[1015]:= HLC_Capture53_TOF.Q;

	(*Fault1016 - IC03OP2 Motion Faults*)
		Fault_Tmrs[1016].PT:=Short_Faults;
		Fault_Tmrs[1016]();
		Fault_Tmrs[1016].IN:= GTAC_CONFIG.Option_HumanFix_Enables.6 AND
							Out_To_ICxx.Fix06_Discrete_Image.CLFaulted.0;
		Out_To_ICxx.System_Faults[1016]:=Fault_Tmrs[1016].Q;
	(*Fault1017 - IC03OP2 Part Present Faults*)
		Fault_Tmrs[1017].PT:=Short_Faults;
		Fault_Tmrs[1017]();
		Fault_Tmrs[1017].IN:= GTAC_CONFIG.Option_HumanFix_Enables.6 AND
							Out_To_ICxx.Fix06_Discrete_Image.PPFaulted.0;
		Out_To_ICxx.System_Faults[1017]:=Fault_Tmrs[1017].Q;
	(*Fault1018 - IC03OP2 Vertical LC Broken While Robot(s) In Zone*)
		VLC_Capture61_TOF.PT:= T#2.0S;
		VLC_Capture61_TOF();
		VLC_Capture61_TOF.IN:= (GTAC_CONFIG.Option_IC_Count>=3) AND GTAC_CONFIG.Option_HumanFix_Enables.6 AND
								NOT MAIN.IC03.OP2_HumanVertLC_Clear AND NOT Fix06.All_Robots_Clear;
		Out_To_ICxx.System_Faults[1018]:= VLC_Capture61_TOF.Q;
	(*Fault1019 - IC03OP2 Horizontal LC Broken While Robot(s) In Zone*)
		HLC_Capture62_TOF.PT:= T#2.0S;
		HLC_Capture62_TOF();
		HLC_Capture62_TOF.IN:= (GTAC_CONFIG.Option_IC_Count>=3) AND GTAC_CONFIG.Option_HumanFix_Enables.6 AND
								NOT MAIN.IC03.OP2_HumanHorizLC_Clear AND NOT Fix06.All_Robots_Clear;
		Out_To_ICxx.System_Faults[1019]:= HLC_Capture62_TOF.Q;
	(*Fault1020 - IC03OP2 Horizontal LC3 Broken While Robot(s) In Zone*)
		HLC_Capture63_TOF.PT:= T#2.0S;
		HLC_Capture63_TOF();
		HLC_Capture63_TOF.IN:= (GTAC_CONFIG.Option_IC_Count>=3) AND GTAC_CONFIG.Option_HumanFix_Enables.6 AND
								NOT MAIN.IC03.OP2_RobotVertLC_Clear AND NOT Fix06.All_Robots_Clear;
		Out_To_ICxx.System_Faults[1020]:= HLC_Capture63_TOF.Q;

	(*------------------- IC04 -----------------*)
	(*Fault1021 - IC04OP1 Motion Faults*)
		Fault_Tmrs[1021].PT:=Short_Faults;
		Fault_Tmrs[1021]();
		Fault_Tmrs[1021].IN:= GTAC_CONFIG.Option_HumanFix_Enables.7 AND
							Out_To_ICxx.Fix07_Discrete_Image.CLFaulted.0;
		Out_To_ICxx.System_Faults[1021]:=Fault_Tmrs[1021].Q;
	(*Fault1022 - IC04OP1 Part Present Faults*)
		Fault_Tmrs[1022].PT:=Short_Faults;
		Fault_Tmrs[1022]();
		Fault_Tmrs[1022].IN:= GTAC_CONFIG.Option_HumanFix_Enables.7 AND
							Out_To_ICxx.Fix07_Discrete_Image.PPFaulted.0;
		Out_To_ICxx.System_Faults[1022]:=Fault_Tmrs[1022].Q;
	(*Fault1023 - IC04OP1 Vertical LC Broken While Robot(s) In Zone*)
		VLC_Capture71_TOF.PT:= T#2.0S;
		VLC_Capture71_TOF();
		VLC_Capture71_TOF.IN:= (GTAC_CONFIG.Option_IC_Count>=4) AND GTAC_CONFIG.Option_HumanFix_Enables.7 AND
								NOT MAIN.IC04.OP1_HumanVertLC_Clear AND NOT Fix07.All_Robots_Clear;
		Out_To_ICxx.System_Faults[1023]:= VLC_Capture71_TOF.Q;
	(*Fault1024 - IC04OP1 Horizontal LC Broken While Robot(s) In Zone*)
		HLC_Capture72_TOF.PT:= T#2.0S;
		HLC_Capture72_TOF();
		HLC_Capture72_TOF.IN:= (GTAC_CONFIG.Option_IC_Count>=4) AND GTAC_CONFIG.Option_HumanFix_Enables.7 AND
								NOT MAIN.IC04.OP1_HumanHorizLC_Clear AND NOT Fix07.All_Robots_Clear;
		Out_To_ICxx.System_Faults[1024]:= HLC_Capture72_TOF.Q;
	(*Fault1025 - IC04OP1 Horizontal LC3 Broken While Robot(s) In Zone*)
		HLC_Capture73_TOF.PT:= T#2.0S;
		HLC_Capture73_TOF();
		HLC_Capture73_TOF.IN:= (GTAC_CONFIG.Option_IC_Count>=4) AND GTAC_CONFIG.Option_HumanFix_Enables.7 AND
								NOT MAIN.IC04.OP1_RobotVertLC_Clear AND NOT Fix07.All_Robots_Clear;
		Out_To_ICxx.System_Faults[1025]:= HLC_Capture73_TOF.Q;

	(*Fault1026 - IC04OP2 Motion Faults*)
		Fault_Tmrs[1026].PT:=Short_Faults;
		Fault_Tmrs[1026]();
		Fault_Tmrs[1026].IN:= GTAC_CONFIG.Option_HumanFix_Enables.8 AND
							Out_To_ICxx.Fix08_Discrete_Image.CLFaulted.0;
		Out_To_ICxx.System_Faults[1026]:=Fault_Tmrs[1026].Q;
	(*Fault1027 - IC04OP2 Part Present Faults*)
		Fault_Tmrs[1027].PT:=Short_Faults;
		Fault_Tmrs[1027]();
		Fault_Tmrs[1027].IN:= GTAC_CONFIG.Option_HumanFix_Enables.8 AND
							Out_To_ICxx.Fix08_Discrete_Image.PPFaulted.0;
		Out_To_ICxx.System_Faults[1027]:=Fault_Tmrs[1027].Q;
	(*Fault1028 - IC04OP2 Vertical LC Broken While Robot(s) In Zone*)
		VLC_Capture81_TOF.PT:= T#2.0S;
		VLC_Capture81_TOF();
		VLC_Capture81_TOF.IN:= (GTAC_CONFIG.Option_IC_Count>=4) AND GTAC_CONFIG.Option_HumanFix_Enables.8 AND
								NOT MAIN.IC04.OP2_HumanVertLC_Clear AND NOT Fix08.All_Robots_Clear;
		Out_To_ICxx.System_Faults[1028]:= VLC_Capture81_TOF.Q;
	(*Fault1029 - IC04OP2 Horizontal LC Broken While Robot(s) In Zone*)
		HLC_Capture82_TOF.PT:= T#2.0S;
		HLC_Capture82_TOF();
		HLC_Capture82_TOF.IN:= (GTAC_CONFIG.Option_IC_Count>=4) AND GTAC_CONFIG.Option_HumanFix_Enables.8 AND
								NOT MAIN.IC04.OP2_HumanHorizLC_Clear AND NOT Fix08.All_Robots_Clear;
		Out_To_ICxx.System_Faults[1029]:= HLC_Capture82_TOF.Q;
	(*Fault1030 - IC04OP2 Horizontal LC3 Broken While Robot(s) In Zone*)
		HLC_Capture83_TOF.PT:= T#2.0S;
		HLC_Capture83_TOF();
		HLC_Capture83_TOF.IN:= (GTAC_CONFIG.Option_IC_Count>=4) AND GTAC_CONFIG.Option_HumanFix_Enables.8 AND
								NOT MAIN.IC04.OP2_RobotVertLC_Clear AND NOT Fix08.All_Robots_Clear;
		Out_To_ICxx.System_Faults[1030]:= HLC_Capture83_TOF.Q;

	(*------------------- IC05 -----------------*)
	(*Fault1031 - IC05OP1 Motion Faults*)
		Fault_Tmrs[1031].PT:=Short_Faults;
		Fault_Tmrs[1031]();
		Fault_Tmrs[1031].IN:= GTAC_CONFIG.Option_HumanFix_Enables.9 AND
							Out_To_ICxx.Fix09_Discrete_Image.CLFaulted.0;
		Out_To_ICxx.System_Faults[1031]:=Fault_Tmrs[1031].Q;
	(*Fault1032 - IC05OP1 Part Present Faults*)
		Fault_Tmrs[1032].PT:=Short_Faults;
		Fault_Tmrs[1032]();
		Fault_Tmrs[1032].IN:= GTAC_CONFIG.Option_HumanFix_Enables.9 AND
							Out_To_ICxx.Fix09_Discrete_Image.PPFaulted.0;
		Out_To_ICxx.System_Faults[1032]:=Fault_Tmrs[1032].Q;
	(*Fault1033 - IC05OP1 Vertical LC Broken While Robot(s) In Zone*)
		VLC_Capture91_TOF.PT:= T#2.0S;
		VLC_Capture91_TOF();
		VLC_Capture91_TOF.IN:= (GTAC_CONFIG.Option_IC_Count>=5) AND GTAC_CONFIG.Option_HumanFix_Enables.9 AND
								NOT MAIN.IC05.OP1_HumanVertLC_Clear AND NOT Fix09.All_Robots_Clear;
		Out_To_ICxx.System_Faults[1033]:= VLC_Capture91_TOF.Q;
	(*Fault1034 - IC05OP1 Horizontal LC Broken While Robot(s) In Zone*)
		HLC_Capture92_TOF.PT:= T#2.0S;
		HLC_Capture92_TOF();
		HLC_Capture92_TOF.IN:= (GTAC_CONFIG.Option_IC_Count>=5) AND GTAC_CONFIG.Option_HumanFix_Enables.9 AND
								NOT MAIN.IC05.OP1_HumanHorizLC_Clear AND NOT Fix09.All_Robots_Clear;
		Out_To_ICxx.System_Faults[1034]:= HLC_Capture92_TOF.Q;
	(*Fault1035 - IC05OP1 Horizontal LC3 Broken While Robot(s) In Zone*)
		HLC_Capture93_TOF.PT:= T#2.0S;
		HLC_Capture93_TOF();
		HLC_Capture93_TOF.IN:= (GTAC_CONFIG.Option_IC_Count>=5) AND GTAC_CONFIG.Option_HumanFix_Enables.9 AND
								NOT MAIN.IC05.OP1_RobotVertLC_Clear AND NOT Fix09.All_Robots_Clear;
		Out_To_ICxx.System_Faults[1035]:= HLC_Capture93_TOF.Q;

	(*Fault1036 - IC05OP2 Motion Faults*)
		Fault_Tmrs[1036].PT:=Short_Faults;
		Fault_Tmrs[1036]();
		Fault_Tmrs[1036].IN:= GTAC_CONFIG.Option_HumanFix_Enables.10 AND
							Out_To_ICxx.Fix10_Discrete_Image.CLFaulted.0;
		Out_To_ICxx.System_Faults[1036]:=Fault_Tmrs[1036].Q;
	(*Fault1037 - IC05OP2 Part Present Faults*)
		Fault_Tmrs[1037].PT:=Short_Faults;
		Fault_Tmrs[1037]();
		Fault_Tmrs[1037].IN:= GTAC_CONFIG.Option_HumanFix_Enables.10 AND
							Out_To_ICxx.Fix10_Discrete_Image.PPFaulted.0;
		Out_To_ICxx.System_Faults[1037]:=Fault_Tmrs[1037].Q;
	(*Fault1038 - IC05OP2 Vertical LC Broken While Robot(s) In Zone*)
		VLC_Capture101_TOF.PT:= T#2.0S;
		VLC_Capture101_TOF();
		VLC_Capture101_TOF.IN:= (GTAC_CONFIG.Option_IC_Count>=5) AND GTAC_CONFIG.Option_HumanFix_Enables.10 AND
									NOT MAIN.IC05.OP2_HumanVertLC_Clear AND NOT Fix10.All_Robots_Clear;
		Out_To_ICxx.System_Faults[1038]:= VLC_Capture101_TOF.Q;
	(*Fault1039 - IC05OP2 Horizontal LC Broken While Robot(s) In Zone*)
		HLC_Capture102_TOF.PT:= T#2.0S;
		HLC_Capture102_TOF();
		HLC_Capture102_TOF.IN:= (GTAC_CONFIG.Option_IC_Count>=5) AND GTAC_CONFIG.Option_HumanFix_Enables.10 AND
									NOT MAIN.IC05.OP2_HumanHorizLC_Clear AND NOT Fix10.All_Robots_Clear;
		Out_To_ICxx.System_Faults[1039]:= HLC_Capture102_TOF.Q;
	(*Fault1040 - IC05OP2 Horizontal LC3 Broken While Robot(s) In Zone*)
		HLC_Capture103_TOF.PT:= T#2.0S;
		HLC_Capture103_TOF();
		HLC_Capture103_TOF.IN:= (GTAC_CONFIG.Option_IC_Count>=5) AND GTAC_CONFIG.Option_HumanFix_Enables.10 AND
									NOT MAIN.IC05.OP2_RobotVertLC_Clear AND NOT Fix10.All_Robots_Clear;
		Out_To_ICxx.System_Faults[1040]:= HLC_Capture103_TOF.Q;

	(*------------------- IC06 -----------------*)
	(*Fault1041 - IC06OP1 Motion Faults*)
		Fault_Tmrs[1041].PT:=Short_Faults;
		Fault_Tmrs[1041]();
		Fault_Tmrs[1041].IN:= GTAC_CONFIG.Option_HumanFix_Enables.11 AND
							Out_To_ICxx.Fix11_Discrete_Image.CLFaulted.0;
		Out_To_ICxx.System_Faults[1041]:=Fault_Tmrs[1041].Q;
	(*Fault1042 - IC06OP1 Part Present Faults*)
		Fault_Tmrs[1042].PT:=Short_Faults;
		Fault_Tmrs[1042]();
		Fault_Tmrs[1042].IN:= GTAC_CONFIG.Option_HumanFix_Enables.11 AND
							Out_To_ICxx.Fix11_Discrete_Image.PPFaulted.0;
		Out_To_ICxx.System_Faults[1042]:=Fault_Tmrs[1042].Q;
	(*Fault1043 - IC06OP1 Vertical LC Broken While Robot(s) In Zone*)
		VLC_Capture111_TOF.PT:= T#2.0S;
		VLC_Capture111_TOF();
		VLC_Capture111_TOF.IN:= (GTAC_CONFIG.Option_IC_Count>=6) AND GTAC_CONFIG.Option_HumanFix_Enables.11 AND
									NOT MAIN.IC06.OP1_HumanVertLC_Clear AND NOT Fix11.All_Robots_Clear;
		Out_To_ICxx.System_Faults[1043]:= VLC_Capture111_TOF.Q;
	(*Fault1044 - IC06OP1 Horizontal LC Broken While Robot(s) In Zone*)
		HLC_Capture112_TOF.PT:= T#2.0S;
		HLC_Capture112_TOF();
		HLC_Capture112_TOF.IN:= (GTAC_CONFIG.Option_IC_Count>=6) AND GTAC_CONFIG.Option_HumanFix_Enables.11 AND
									NOT MAIN.IC06.OP1_HumanHorizLC_Clear AND NOT Fix11.All_Robots_Clear;
		Out_To_ICxx.System_Faults[1044]:= HLC_Capture112_TOF.Q;
	(*Fault1045 - IC06OP1 Horizontal LC3 Broken While Robot(s) In Zone*)
		HLC_Capture113_TOF.PT:= T#2.0S;
		HLC_Capture113_TOF();
		HLC_Capture113_TOF.IN:= (GTAC_CONFIG.Option_IC_Count>=6) AND GTAC_CONFIG.Option_HumanFix_Enables.11 AND
									NOT MAIN.IC06.OP1_RobotVertLC_Clear AND NOT Fix11.All_Robots_Clear;
		Out_To_ICxx.System_Faults[1045]:= HLC_Capture113_TOF.Q;

	(*Fault1046 - IC06OP2 Motion Faults*)
		Fault_Tmrs[1046].PT:=Short_Faults;
		Fault_Tmrs[1046]();
		Fault_Tmrs[1046].IN:= GTAC_CONFIG.Option_HumanFix_Enables.12 AND
							Out_To_ICxx.Fix12_Discrete_Image.CLFaulted.0;
		Out_To_ICxx.System_Faults[1046]:=Fault_Tmrs[1046].Q;
	(*Fault1047 - IC06OP2 Part Present Faults*)
		Fault_Tmrs[1047].PT:=Short_Faults;
		Fault_Tmrs[1047]();
		Fault_Tmrs[1047].IN:= GTAC_CONFIG.Option_HumanFix_Enables.12 AND
							Out_To_ICxx.Fix12_Discrete_Image.PPFaulted.0;
		Out_To_ICxx.System_Faults[1047]:=Fault_Tmrs[1047].Q;
	(*Fault1048 - IC06OP2 Vertical LC Broken While Robot(s) In Zone*)
		VLC_Capture121_TOF.PT:= T#2.0S;
		VLC_Capture121_TOF();
		VLC_Capture121_TOF.IN:= (GTAC_CONFIG.Option_IC_Count>=6) AND GTAC_CONFIG.Option_HumanFix_Enables.12 AND
									NOT MAIN.IC06.OP2_HumanVertLC_Clear AND NOT Fix12.All_Robots_Clear;
		Out_To_ICxx.System_Faults[1048]:= VLC_Capture121_TOF.Q;
	(*Fault1049 - IC06OP2 Horizontal LC Broken While Robot(s) In Zone*)
		HLC_Capture122_TOF.PT:= T#2.0S;
		HLC_Capture122_TOF();
		HLC_Capture122_TOF.IN:= (GTAC_CONFIG.Option_IC_Count>=6) AND GTAC_CONFIG.Option_HumanFix_Enables.12 AND
									NOT MAIN.IC06.OP2_HumanHorizLC_Clear AND NOT Fix12.All_Robots_Clear;
		Out_To_ICxx.System_Faults[1049]:= HLC_Capture122_TOF.Q;
	(*Fault1050 - IC06OP2 Horizontal LC3 Broken While Robot(s) In Zone*)
		HLC_Capture123_TOF.PT:= T#2.0S;
		HLC_Capture123_TOF();
		HLC_Capture123_TOF.IN:= (GTAC_CONFIG.Option_IC_Count>=6) AND GTAC_CONFIG.Option_HumanFix_Enables.12 AND
									NOT MAIN.IC06.OP2_RobotVertLC_Clear AND NOT Fix12.All_Robots_Clear;
		Out_To_ICxx.System_Faults[1050]:= HLC_Capture123_TOF.Q;

	(*------------------- IC07 -----------------*)
	(*Fault1051 - IC07OP1 Motion Faults*)
		Fault_Tmrs[1051].PT:=Short_Faults;
		Fault_Tmrs[1051]();
		Fault_Tmrs[1051].IN:= GTAC_CONFIG.Option_HumanFix_Enables.13 AND
							Out_To_ICxx.Fix13_Discrete_Image.CLFaulted.0;
		Out_To_ICxx.System_Faults[1051]:=Fault_Tmrs[1051].Q;
	(*Fault1052 - IC07OP1 Part Present Faults*)
		Fault_Tmrs[1052].PT:=Short_Faults;
		Fault_Tmrs[1052]();
		Fault_Tmrs[1052].IN:= GTAC_CONFIG.Option_HumanFix_Enables.13 AND
							Out_To_ICxx.Fix13_Discrete_Image.PPFaulted.0;
		Out_To_ICxx.System_Faults[1052]:=Fault_Tmrs[1052].Q;
	(*Fault1053 - IC07OP1 Vertical LC Broken While Robot(s) In Zone*)
		VLC_Capture131_TOF.PT:= T#2.0S;
		VLC_Capture131_TOF();
		VLC_Capture131_TOF.IN:= (GTAC_CONFIG.Option_IC_Count>=7) AND GTAC_CONFIG.Option_HumanFix_Enables.13 AND
									NOT MAIN.IC07.OP1_HumanVertLC_Clear AND NOT Fix13.All_Robots_Clear;
		Out_To_ICxx.System_Faults[1053]:= VLC_Capture131_TOF.Q;
	(*Fault1054 - IC07OP1 Horizontal LC Broken While Robot(s) In Zone*)
		HLC_Capture132_TOF.PT:= T#2.0S;
		HLC_Capture132_TOF();
		HLC_Capture132_TOF.IN:= (GTAC_CONFIG.Option_IC_Count>=7) AND GTAC_CONFIG.Option_HumanFix_Enables.13 AND
									NOT MAIN.IC07.OP1_HumanHorizLC_Clear AND NOT Fix13.All_Robots_Clear;
		Out_To_ICxx.System_Faults[1054]:= HLC_Capture132_TOF.Q;
	(*Fault1055 - IC07OP1 Horizontal LC3 Broken While Robot(s) In Zone*)
		HLC_Capture133_TOF.PT:= T#2.0S;
		HLC_Capture133_TOF();
		HLC_Capture133_TOF.IN:= (GTAC_CONFIG.Option_IC_Count>=7) AND GTAC_CONFIG.Option_HumanFix_Enables.13 AND
									NOT MAIN.IC07.OP1_RobotVertLC_Clear AND NOT Fix13.All_Robots_Clear;
		Out_To_ICxx.System_Faults[1055]:= HLC_Capture133_TOF.Q;

	(*Fault1056 - IC07OP2 Motion Faults*)
		Fault_Tmrs[1056].PT:=Short_Faults;
		Fault_Tmrs[1056]();
		Fault_Tmrs[1056].IN:= GTAC_CONFIG.Option_HumanFix_Enables.14 AND
							Out_To_ICxx.Fix14_Discrete_Image.CLFaulted.0;
		Out_To_ICxx.System_Faults[1056]:=Fault_Tmrs[1056].Q;
	(*Fault1057 - IC07OP2 Part Present Faults*)
		Fault_Tmrs[1057].PT:=Short_Faults;
		Fault_Tmrs[1057]();
		Fault_Tmrs[1057].IN:= GTAC_CONFIG.Option_HumanFix_Enables.14 AND
							Out_To_ICxx.Fix14_Discrete_Image.PPFaulted.0;
		Out_To_ICxx.System_Faults[1057]:=Fault_Tmrs[1057].Q;
	(*Fault1058 - IC07OP2 Vertical LC Broken While Robot(s) In Zone*)
		VLC_Capture141_TOF.PT:= T#2.0S;
		VLC_Capture141_TOF();
		VLC_Capture141_TOF.IN:= (GTAC_CONFIG.Option_IC_Count>=7) AND GTAC_CONFIG.Option_HumanFix_Enables.14 AND
									NOT MAIN.IC07.OP2_HumanVertLC_Clear AND NOT Fix14.All_Robots_Clear;
		Out_To_ICxx.System_Faults[1058]:= VLC_Capture141_TOF.Q;
	(*Fault1059 - IC07OP2 Horizontal LC Broken While Robot(s) In Zone*)
		HLC_Capture142_TOF.PT:= T#2.0S;
		HLC_Capture142_TOF();
		HLC_Capture142_TOF.IN:= (GTAC_CONFIG.Option_IC_Count>=7) AND GTAC_CONFIG.Option_HumanFix_Enables.14 AND
									NOT MAIN.IC07.OP2_HumanHorizLC_Clear AND NOT Fix14.All_Robots_Clear;
		Out_To_ICxx.System_Faults[1059]:= HLC_Capture142_TOF.Q;
	(*Fault1060 - IC07OP2 Horizontal LC3 Broken While Robot(s) In Zone*)
		HLC_Capture143_TOF.PT:= T#2.0S;
		HLC_Capture143_TOF();
		HLC_Capture143_TOF.IN:= (GTAC_CONFIG.Option_IC_Count>=7) AND GTAC_CONFIG.Option_HumanFix_Enables.14 AND
									NOT MAIN.IC07.OP2_RobotVertLC_Clear AND NOT Fix14.All_Robots_Clear;
		Out_To_ICxx.System_Faults[1060]:= HLC_Capture143_TOF.Q;

	(*------------------- IC08 -----------------*)
	(*Fault1061 - IC08OP1 Motion Faults*)
		Fault_Tmrs[1061].PT:=Short_Faults;
		Fault_Tmrs[1061]();
		Fault_Tmrs[1061].IN:= GTAC_CONFIG.Option_HumanFix_Enables.15 AND
							Out_To_ICxx.Fix15_Discrete_Image.CLFaulted.0;
		Out_To_ICxx.System_Faults[1061]:=Fault_Tmrs[1061].Q;
	(*Fault1062 - IC08OP1 Part Present Faults*)
		Fault_Tmrs[1062].PT:=Short_Faults;
		Fault_Tmrs[1062]();
		Fault_Tmrs[1062].IN:= GTAC_CONFIG.Option_HumanFix_Enables.15 AND
							Out_To_ICxx.Fix15_Discrete_Image.PPFaulted.0;
		Out_To_ICxx.System_Faults[1062]:=Fault_Tmrs[1062].Q;
	(*Fault1063 - IC08OP1 Vertical LC Broken While Robot(s) In Zone*)
		VLC_Capture151_TOF.PT:= T#2.0S;
		VLC_Capture151_TOF();
		VLC_Capture151_TOF.IN:= (GTAC_CONFIG.Option_IC_Count>=8) AND GTAC_CONFIG.Option_HumanFix_Enables.15 AND
									NOT MAIN.IC08.OP1_HumanVertLC_Clear AND NOT Fix15.All_Robots_Clear;
		Out_To_ICxx.System_Faults[1063]:= VLC_Capture151_TOF.Q;
	(*Fault1064 - IC08OP1 Horizontal LC Broken While Robot(s) In Zone*)
		HLC_Capture152_TOF.PT:= T#2.0S;
		HLC_Capture152_TOF();
		HLC_Capture152_TOF.IN:= (GTAC_CONFIG.Option_IC_Count>=8) AND GTAC_CONFIG.Option_HumanFix_Enables.15 AND
									NOT MAIN.IC08.OP1_HumanHorizLC_Clear AND NOT Fix15.All_Robots_Clear;
		Out_To_ICxx.System_Faults[1064]:= HLC_Capture152_TOF.Q;
	(*Fault1065 - IC08OP1 Horizontal LC3 Broken While Robot(s) In Zone*)
		HLC_Capture153_TOF.PT:= T#2.0S;
		HLC_Capture153_TOF();
		HLC_Capture153_TOF.IN:= (GTAC_CONFIG.Option_IC_Count>=8) AND GTAC_CONFIG.Option_HumanFix_Enables.15 AND
									NOT MAIN.IC08.OP1_RobotVertLC_Clear AND NOT Fix15.All_Robots_Clear;
		Out_To_ICxx.System_Faults[1065]:= HLC_Capture153_TOF.Q;

	(*Fault1066 - IC08OP2 Motion Faults*)
		Fault_Tmrs[1066].PT:=Short_Faults;
		Fault_Tmrs[1066]();
		Fault_Tmrs[1066].IN:= GTAC_CONFIG.Option_HumanFix_Enables.16 AND
							Out_To_ICxx.Fix16_Discrete_Image.CLFaulted.0;
		Out_To_ICxx.System_Faults[1066]:=Fault_Tmrs[1066].Q;
	(*Fault1067 - IC08OP2 Part Present Faults*)
		Fault_Tmrs[1067].PT:=Short_Faults;
		Fault_Tmrs[1067]();
		Fault_Tmrs[1067].IN:= GTAC_CONFIG.Option_HumanFix_Enables.16 AND
							Out_To_ICxx.Fix16_Discrete_Image.PPFaulted.0;
		Out_To_ICxx.System_Faults[1067]:=Fault_Tmrs[1067].Q;
	(*Fault1068 - IC08OP2 Vertical LC Broken While Robot(s) In Zone*)
		VLC_Capture161_TOF.PT:= T#2.0S;
		VLC_Capture161_TOF();
		VLC_Capture161_TOF.IN:= (GTAC_CONFIG.Option_IC_Count>=8) AND GTAC_CONFIG.Option_HumanFix_Enables.16 AND
									NOT MAIN.IC08.OP2_HumanVertLC_Clear AND NOT Fix16.All_Robots_Clear;
		Out_To_ICxx.System_Faults[1068]:= VLC_Capture161_TOF.Q;
	(*Fault1069 - IC08OP2 Horizontal LC Broken While Robot(s) In Zone*)
		HLC_Capture162_TOF.PT:= T#2.0S;
		HLC_Capture162_TOF();
		HLC_Capture162_TOF.IN:= (GTAC_CONFIG.Option_IC_Count>=8) AND GTAC_CONFIG.Option_HumanFix_Enables.16 AND
									NOT MAIN.IC08.OP2_HumanHorizLC_Clear AND NOT Fix16.All_Robots_Clear;
		Out_To_ICxx.System_Faults[1069]:= HLC_Capture162_TOF.Q;
	(*Fault1070 - IC08OP2 Horizontal LC3 Broken While Robot(s) In Zone*)
		HLC_Capture163_TOF.PT:= T#2.0S;
		HLC_Capture163_TOF();
		HLC_Capture163_TOF.IN:= (GTAC_CONFIG.Option_IC_Count>=8) AND GTAC_CONFIG.Option_HumanFix_Enables.16 AND
									NOT MAIN.IC08.OP2_RobotVertLC_Clear AND NOT Fix16.All_Robots_Clear;
		Out_To_ICxx.System_Faults[1070]:= HLC_Capture163_TOF.Q;

	(*--------------------------------------------------------------------------- Internal Fixture Faults--------------------------------------------------------------------*)
	(*Fault1071 - Fix101 Motion Faults*)
		Fault_Tmrs[1071].PT:=Short_Faults;
		Fault_Tmrs[1071]();
		Fault_Tmrs[1071].IN:= (GTAC_CONFIG.Option_InternalFix_Count>=1)  AND
							Out_To_ICxx.Fix101_Discrete_Image.CLFaulted.0;
		Out_To_ICxx.System_Faults[1071]:=Fault_Tmrs[1071].Q;
	(*Fault1072 - Fix101 Part Present Faults*)
		Fault_Tmrs[1072].PT:=Short_Faults;
		Fault_Tmrs[1072]();
		Fault_Tmrs[1072].IN:= (GTAC_CONFIG.Option_InternalFix_Count>=1)  AND
							Out_To_ICxx.Fix101_Discrete_Image.PPFaulted.0;
		Out_To_ICxx.System_Faults[1072]:=Fault_Tmrs[1072].Q;

	(*Fault1074 - Fix102 Motion Faults*)
		Fault_Tmrs[1074].PT:=Short_Faults;
		Fault_Tmrs[1074]();
		Fault_Tmrs[1074].IN:= (GTAC_CONFIG.Option_InternalFix_Count>=2)  AND
							Out_To_ICxx.Fix102_Discrete_Image.CLFaulted.0;
		Out_To_ICxx.System_Faults[1074]:=Fault_Tmrs[1074].Q;
	(*Fault1075 - Fix102 Part Present Faults*)
		Fault_Tmrs[1075].PT:=Short_Faults;
		Fault_Tmrs[1075]();
		Fault_Tmrs[1075].IN:= (GTAC_CONFIG.Option_InternalFix_Count>=2)  AND
							Out_To_ICxx.Fix102_Discrete_Image.PPFaulted.0;
		Out_To_ICxx.System_Faults[1075]:=Fault_Tmrs[1075].Q;

	(*Fault1077 - Fix103 Motion Faults*)
		Fault_Tmrs[1077].PT:=Short_Faults;
		Fault_Tmrs[1077]();
		Fault_Tmrs[1077].IN:= (GTAC_CONFIG.Option_InternalFix_Count>=3)  AND
							Out_To_ICxx.Fix103_Discrete_Image.CLFaulted.0;
		Out_To_ICxx.System_Faults[1077]:=Fault_Tmrs[1077].Q;
	(*Fault1078 - Fix103 Part Present Faults*)
		Fault_Tmrs[1078].PT:=Short_Faults;
		Fault_Tmrs[1078]();
		Fault_Tmrs[1078].IN:= (GTAC_CONFIG.Option_InternalFix_Count>=3)  AND
							Out_To_ICxx.Fix103_Discrete_Image.PPFaulted.0;
		Out_To_ICxx.System_Faults[1078]:=Fault_Tmrs[1078].Q;

	(*Fault1080 - Fix104 Motion Faults*)
		Fault_Tmrs[1080].PT:=Short_Faults;
		Fault_Tmrs[1080]();
		Fault_Tmrs[1080].IN:= (GTAC_CONFIG.Option_InternalFix_Count>=4)  AND
							Out_To_ICxx.Fix104_Discrete_Image.CLFaulted.0;
		Out_To_ICxx.System_Faults[1080]:=Fault_Tmrs[1080].Q;
	(*Fault1081 - Fix104 Part Present Faults*)
		Fault_Tmrs[1081].PT:=Short_Faults;
		Fault_Tmrs[1081]();
		Fault_Tmrs[1081].IN:= (GTAC_CONFIG.Option_InternalFix_Count>=4)  AND
							Out_To_ICxx.Fix104_Discrete_Image.PPFaulted.0;
		Out_To_ICxx.System_Faults[1081]:=Fault_Tmrs[1081].Q;

	(*Fault1083 - Fix105 Motion Faults*)
		Fault_Tmrs[1083].PT:=Short_Faults;
		Fault_Tmrs[1083]();
		Fault_Tmrs[1083].IN:= (GTAC_CONFIG.Option_InternalFix_Count>=5)  AND
							Out_To_ICxx.Fix105_Discrete_Image.CLFaulted.0;
		Out_To_ICxx.System_Faults[1083]:=Fault_Tmrs[1083].Q;
	(*Fault1084 - Fix105 Part Present Faults*)
		Fault_Tmrs[1084].PT:=Short_Faults;
		Fault_Tmrs[1084]();
		Fault_Tmrs[1084].IN:= (GTAC_CONFIG.Option_InternalFix_Count>=5)  AND
							Out_To_ICxx.Fix105_Discrete_Image.PPFaulted.0;
		Out_To_ICxx.System_Faults[1084]:=Fault_Tmrs[1084].Q;

	(*Fault1086 - Fix106 Motion Faults*)
		Fault_Tmrs[1086].PT:=Short_Faults;
		Fault_Tmrs[1086]();
		Fault_Tmrs[1086].IN:= (GTAC_CONFIG.Option_InternalFix_Count>=6)  AND
							Out_To_ICxx.Fix106_Discrete_Image.CLFaulted.0;
		Out_To_ICxx.System_Faults[1086]:=Fault_Tmrs[1086].Q;
	(*Fault1087 - Fix106 Part Present Faults*)
		Fault_Tmrs[1087].PT:=Short_Faults;
		Fault_Tmrs[1087]();
		Fault_Tmrs[1087].IN:= (GTAC_CONFIG.Option_InternalFix_Count>=6)  AND
							Out_To_ICxx.Fix106_Discrete_Image.PPFaulted.0;
		Out_To_ICxx.System_Faults[1087]:=Fault_Tmrs[1087].Q;

	(*Fault1089 - Fix107 Motion Faults*)
		Fault_Tmrs[1089].PT:=Short_Faults;
		Fault_Tmrs[1089]();
		Fault_Tmrs[1089].IN:= (GTAC_CONFIG.Option_InternalFix_Count>=7)  AND
							Out_To_ICxx.Fix107_Discrete_Image.CLFaulted.0;
		Out_To_ICxx.System_Faults[1089]:=Fault_Tmrs[1089].Q;
	(*Fault1090 - Fix107 Part Present Faults*)
		Fault_Tmrs[1090].PT:=Short_Faults;
		Fault_Tmrs[1090]();
		Fault_Tmrs[1090].IN:= (GTAC_CONFIG.Option_InternalFix_Count>=7)  AND
							Out_To_ICxx.Fix107_Discrete_Image.PPFaulted.0;
		Out_To_ICxx.System_Faults[1090]:=Fault_Tmrs[1090].Q;

	(*Fault1092 - Fix108 Motion Faults*)
		Fault_Tmrs[1092].PT:=Short_Faults;
		Fault_Tmrs[1092]();
		Fault_Tmrs[1092].IN:= (GTAC_CONFIG.Option_InternalFix_Count>=8)  AND
							Out_To_ICxx.Fix108_Discrete_Image.CLFaulted.0;
		Out_To_ICxx.System_Faults[1092]:=Fault_Tmrs[1092].Q;
	(*Fault1093 - Fix108 Part Present Faults*)
		Fault_Tmrs[1093].PT:=Short_Faults;
		Fault_Tmrs[1093]();
		Fault_Tmrs[1093].IN:= (GTAC_CONFIG.Option_InternalFix_Count>=8)  AND
							Out_To_ICxx.Fix108_Discrete_Image.PPFaulted.0;
		Out_To_ICxx.System_Faults[1093]:=Fault_Tmrs[1093].Q;

	(*Fault1095 - Fix109 Motion Faults*)
		Fault_Tmrs[1095].PT:=Short_Faults;
		Fault_Tmrs[1095]();
		Fault_Tmrs[1095].IN:= (GTAC_CONFIG.Option_InternalFix_Count>=9)  AND
							Out_To_ICxx.Fix109_Discrete_Image.CLFaulted.0;
		Out_To_ICxx.System_Faults[1095]:=Fault_Tmrs[1095].Q;
	(*Fault1096 - Fix109 Part Present Faults*)
		Fault_Tmrs[1096].PT:=Short_Faults;
		Fault_Tmrs[1096]();
		Fault_Tmrs[1096].IN:= (GTAC_CONFIG.Option_InternalFix_Count>=9)  AND
							Out_To_ICxx.Fix109_Discrete_Image.PPFaulted.0;
		Out_To_ICxx.System_Faults[1096]:=Fault_Tmrs[1096].Q;

	(*Fault1098 - Fix110 Motion Faults*)
		Fault_Tmrs[1098].PT:=Short_Faults;
		Fault_Tmrs[1098]();
		Fault_Tmrs[1098].IN:= (GTAC_CONFIG.Option_InternalFix_Count>=10)  AND
							Out_To_ICxx.Fix110_Discrete_Image.CLFaulted.0;
		Out_To_ICxx.System_Faults[1098]:=Fault_Tmrs[1098].Q;
	(*Fault1099 - Fix110 Part Present Faults*)
		Fault_Tmrs[1099].PT:=Short_Faults;
		Fault_Tmrs[1099]();
		Fault_Tmrs[1099].IN:= (GTAC_CONFIG.Option_InternalFix_Count>=10)  AND
							Out_To_ICxx.Fix110_Discrete_Image.PPFaulted.0;
		Out_To_ICxx.System_Faults[1099]:=Fault_Tmrs[1099].Q;

	(*Fault1101 - Fix111 Motion Faults*)
		Fault_Tmrs[1101].PT:=Short_Faults;
		Fault_Tmrs[1101]();
		Fault_Tmrs[1101].IN:= (GTAC_CONFIG.Option_InternalFix_Count>=11)  AND
							Out_To_ICxx.Fix111_Discrete_Image.CLFaulted.0;
		Out_To_ICxx.System_Faults[1101]:=Fault_Tmrs[1101].Q;
	(*Fault1102 - Fix111 Part Present Faults*)
		Fault_Tmrs[1102].PT:=Short_Faults;
		Fault_Tmrs[1102]();
		Fault_Tmrs[1102].IN:= (GTAC_CONFIG.Option_InternalFix_Count>=11)  AND
							Out_To_ICxx.Fix111_Discrete_Image.PPFaulted.0;
		Out_To_ICxx.System_Faults[1102]:=Fault_Tmrs[1102].Q;
	
	(*Fault1104 - Fix112 Motion Faults*)
		Fault_Tmrs[1104].PT:=Short_Faults;
		Fault_Tmrs[1104]();
		Fault_Tmrs[1104].IN:= (GTAC_CONFIG.Option_InternalFix_Count>=12)  AND
							Out_To_ICxx.Fix112_Discrete_Image.CLFaulted.0;
		Out_To_ICxx.System_Faults[1104]:=Fault_Tmrs[1104].Q;
	(*Fault1105 - Fix112 Part Present Faults*)
		Fault_Tmrs[1105].PT:=Short_Faults;
		Fault_Tmrs[1105]();
		Fault_Tmrs[1105].IN:= (GTAC_CONFIG.Option_InternalFix_Count>=12)  AND
							Out_To_ICxx.Fix112_Discrete_Image.PPFaulted.0;
		Out_To_ICxx.System_Faults[1105]:=Fault_Tmrs[1105].Q;

	(*----------------------------------------------------------------------------- Robot Faults ------------------------------------------------------------------------------*)
	(*Fault1121 - R1 System Fault*)
		Fault_Tmrs[1121].PT:=Short_Faults;
		Fault_Tmrs[1121]();
		Fault_Tmrs[1121].IN:= (GTAC_CONFIG.Option_Robot_Count>=1) AND
							(MAIN.R1.Battery_Alarm OR (MAIN.R1.Faulted AND MAIN.Control_Power_ON));
		Out_To_ICxx.System_Faults[1121]:=Fault_Tmrs[1121].Q;
	(*Fault1122 - R2 System Fault*)
		Fault_Tmrs[1122].PT:=Short_Faults;
		Fault_Tmrs[1122]();
		Fault_Tmrs[1122].IN:= (GTAC_CONFIG.Option_Robot_Count>=2) AND
							(MAIN.R2.Battery_Alarm OR (MAIN.R2.Faulted AND MAIN.Control_Power_ON));
		Out_To_ICxx.System_Faults[1122]:=Fault_Tmrs[1122].Q;
	(*Fault1123 - R3 System Fault*)
		Fault_Tmrs[1123].PT:=Short_Faults;
		Fault_Tmrs[1123]();
		Fault_Tmrs[1123].IN:= (GTAC_CONFIG.Option_Robot_Count>=3) AND
							(MAIN.R3.Battery_Alarm OR (MAIN.R3.Faulted AND MAIN.Control_Power_ON));
		Out_To_ICxx.System_Faults[1123]:=Fault_Tmrs[1123].Q;
	(*Fault1124 - R4 System Fault*)
		Fault_Tmrs[1124].PT:=Short_Faults;
		Fault_Tmrs[1124]();
		Fault_Tmrs[1124].IN:= (GTAC_CONFIG.Option_Robot_Count>=4) AND
							(MAIN.R4.Battery_Alarm OR (MAIN.R4.Faulted AND MAIN.Control_Power_ON));
		Out_To_ICxx.System_Faults[1124]:=Fault_Tmrs[1124].Q;
	(*Fault1125 - R5 System Fault*)
		Fault_Tmrs[1125].PT:=Short_Faults;
		Fault_Tmrs[1125]();
		Fault_Tmrs[1125].IN:= (GTAC_CONFIG.Option_Robot_Count>=5) AND
							(MAIN.R5.Battery_Alarm OR (MAIN.R5.Faulted AND MAIN.Control_Power_ON));
		Out_To_ICxx.System_Faults[1125]:=Fault_Tmrs[1125].Q;
	(*Fault1126 - R6 System Fault*)
		Fault_Tmrs[1126].PT:=Short_Faults;
		Fault_Tmrs[1126]();
		Fault_Tmrs[1126].IN:= (GTAC_CONFIG.Option_Robot_Count>=6) AND
							(MAIN.R6.Battery_Alarm OR (MAIN.R6.Faulted AND MAIN.Control_Power_ON));
		Out_To_ICxx.System_Faults[1126]:=Fault_Tmrs[1126].Q;
	(*Fault1127 - R7 System Fault*)
		Fault_Tmrs[1127].PT:=Short_Faults;
		Fault_Tmrs[1127]();
		Fault_Tmrs[1127].IN:= (GTAC_CONFIG.Option_Robot_Count>=7) AND
							(MAIN.R7.Battery_Alarm OR (MAIN.R7.Faulted AND MAIN.Control_Power_ON));
		Out_To_ICxx.System_Faults[1127]:=Fault_Tmrs[1127].Q;
	(*Fault1128 - R8 System Fault*)
		Fault_Tmrs[1128].PT:=Short_Faults;
		Fault_Tmrs[1128]();
		Fault_Tmrs[1128].IN:= (GTAC_CONFIG.Option_Robot_Count>=8) AND
							(MAIN.R8.Battery_Alarm OR (MAIN.R8.Faulted AND MAIN.Control_Power_ON));
		Out_To_ICxx.System_Faults[1128]:=Fault_Tmrs[1128].Q;
	(*Fault1129 - R9 System Fault*)
		Fault_Tmrs[1129].PT:=Short_Faults;
		Fault_Tmrs[1129]();
		Fault_Tmrs[1129].IN:= (GTAC_CONFIG.Option_Robot_Count>=9) AND
							(MAIN.R9.Battery_Alarm OR (MAIN.R9.Faulted AND MAIN.Control_Power_ON));
		Out_To_ICxx.System_Faults[1129]:=Fault_Tmrs[1129].Q;
	(*Fault1130 - R10 System Fault*)
		Fault_Tmrs[1130].PT:=Short_Faults;
		Fault_Tmrs[1130]();
		Fault_Tmrs[1130].IN:= (GTAC_CONFIG.Option_Robot_Count>=10) AND
							(MAIN.R10.Battery_Alarm OR (MAIN.R10.Faulted AND MAIN.Control_Power_ON));
		Out_To_ICxx.System_Faults[1130]:=Fault_Tmrs[1130].Q;
	(*Fault1131 - R11 System Fault*)
		Fault_Tmrs[1131].PT:=Short_Faults;
		Fault_Tmrs[1131]();
		Fault_Tmrs[1131].IN:= (GTAC_CONFIG.Option_Robot_Count>=11) AND
							(MAIN.R11.Battery_Alarm OR (MAIN.R11.Faulted AND MAIN.Control_Power_ON));
		Out_To_ICxx.System_Faults[1131]:=Fault_Tmrs[1131].Q;
	(*Fault1132 - R12 System Fault*)
		Fault_Tmrs[1132].PT:=Short_Faults;
		Fault_Tmrs[1132]();
		Fault_Tmrs[1132].IN:= (GTAC_CONFIG.Option_Robot_Count>=12) AND
							(MAIN.R12.Battery_Alarm OR (MAIN.R12.Faulted AND MAIN.Control_Power_ON));
		Out_To_ICxx.System_Faults[1132]:=Fault_Tmrs[1132].Q;
	(*Fault1133 - R13 System Fault*)
		Fault_Tmrs[1133].PT:=Short_Faults;
		Fault_Tmrs[1133]();
		Fault_Tmrs[1133].IN:= (GTAC_CONFIG.Option_Robot_Count>=13) AND
							(MAIN.R13.Battery_Alarm OR (MAIN.R13.Faulted AND MAIN.Control_Power_ON));
		Out_To_ICxx.System_Faults[1133]:=Fault_Tmrs[1133].Q;
	(*Fault1134 - R14 System Fault*)
		Fault_Tmrs[1134].PT:=Short_Faults;
		Fault_Tmrs[1134]();
		Fault_Tmrs[1134].IN:= (GTAC_CONFIG.Option_Robot_Count>=14) AND
							(MAIN.R14.Battery_Alarm OR (MAIN.R14.Faulted AND MAIN.Control_Power_ON));
		Out_To_ICxx.System_Faults[1134]:=Fault_Tmrs[1134].Q;
	(*Fault1135 - R15 System Fault*)
		Fault_Tmrs[1135].PT:=Short_Faults;
		Fault_Tmrs[1135]();
		Fault_Tmrs[1135].IN:= (GTAC_CONFIG.Option_Robot_Count>=15) AND
							(MAIN.R15.Battery_Alarm OR (MAIN.R15.Faulted AND MAIN.Control_Power_ON));
		Out_To_ICxx.System_Faults[1135]:=Fault_Tmrs[1135].Q;
	(*Fault1136 - R16 System Fault*)
		Fault_Tmrs[1136].PT:=Short_Faults;
		Fault_Tmrs[1136]();
		Fault_Tmrs[1136].IN:= (GTAC_CONFIG.Option_Robot_Count>=16) AND
							(MAIN.R16.Battery_Alarm OR (MAIN.R16.Faulted AND MAIN.Control_Power_ON));
		Out_To_ICxx.System_Faults[1136]:=Fault_Tmrs[1136].Q;
	(*Fault1137 - R17 System Fault*)
		Fault_Tmrs[1137].PT:=Short_Faults;
		Fault_Tmrs[1137]();
		Fault_Tmrs[1137].IN:= (GTAC_CONFIG.Option_Robot_Count>=17) AND
							(MAIN.R17.Battery_Alarm OR (MAIN.R17.Faulted AND MAIN.Control_Power_ON));
		Out_To_ICxx.System_Faults[1137]:=Fault_Tmrs[1137].Q;
	(*Fault1138 - R18 System Fault*)
		Fault_Tmrs[1138].PT:=Short_Faults;
		Fault_Tmrs[1138]();
		Fault_Tmrs[1138].IN:= (GTAC_CONFIG.Option_Robot_Count>=18) AND
							(MAIN.R18.Battery_Alarm OR (MAIN.R18.Faulted AND MAIN.Control_Power_ON));
		Out_To_ICxx.System_Faults[1138]:=Fault_Tmrs[1138].Q;
	(*Fault1139 - R19 System Fault*)
		Fault_Tmrs[1139].PT:=Short_Faults;
		Fault_Tmrs[1139]();
		Fault_Tmrs[1139].IN:= (GTAC_CONFIG.Option_Robot_Count>=19) AND
							(MAIN.R19.Battery_Alarm OR (MAIN.R19.Faulted AND MAIN.Control_Power_ON));
		Out_To_ICxx.System_Faults[1139]:=Fault_Tmrs[1139].Q;
	(*Fault1140 - R20 System Fault*)
		Fault_Tmrs[1140].PT:=Short_Faults;
		Fault_Tmrs[1140]();
		Fault_Tmrs[1140].IN:= (GTAC_CONFIG.Option_Robot_Count>=20) AND
							(MAIN.R20.Battery_Alarm OR (MAIN.R20.Faulted AND MAIN.Control_Power_ON));
		Out_To_ICxx.System_Faults[1140]:=Fault_Tmrs[1140].Q;
	(*Fault1141 - R21 System Fault*)
		Fault_Tmrs[1141].PT:=Short_Faults;
		Fault_Tmrs[1141]();
		Fault_Tmrs[1141].IN:= (GTAC_CONFIG.Option_Robot_Count>=21) AND
							(MAIN.R21.Battery_Alarm OR (MAIN.R21.Faulted AND MAIN.Control_Power_ON));
		Out_To_ICxx.System_Faults[1141]:=Fault_Tmrs[1141].Q;
	(*Fault1142 - R22 System Fault*)
		Fault_Tmrs[1142].PT:=Short_Faults;
		Fault_Tmrs[1142]();
		Fault_Tmrs[1142].IN:= (GTAC_CONFIG.Option_Robot_Count>=22) AND
							(MAIN.R22.Battery_Alarm OR (MAIN.R22.Faulted AND MAIN.Control_Power_ON));
		Out_To_ICxx.System_Faults[1142]:=Fault_Tmrs[1142].Q;
	(*Fault1143 - R23 System Fault*)
		Fault_Tmrs[1143].PT:=Short_Faults;
		Fault_Tmrs[1143]();
		Fault_Tmrs[1143].IN:= (GTAC_CONFIG.Option_Robot_Count>=23) AND
							(MAIN.R23.Battery_Alarm OR (MAIN.R23.Faulted AND MAIN.Control_Power_ON));
		Out_To_ICxx.System_Faults[1143]:=Fault_Tmrs[1143].Q;
	(*Fault1144 - R24 System Fault*)
		Fault_Tmrs[1144].PT:=Short_Faults;
		Fault_Tmrs[1144]();
		Fault_Tmrs[1144].IN:= (GTAC_CONFIG.Option_Robot_Count>=24) AND
							(MAIN.R24.Battery_Alarm OR (MAIN.R24.Faulted AND MAIN.Control_Power_ON));
		Out_To_ICxx.System_Faults[1144]:=Fault_Tmrs[1144].Q;
	(*Fault1145 - R25 System Fault*)
		Fault_Tmrs[1145].PT:=Short_Faults;
		Fault_Tmrs[1145]();
		Fault_Tmrs[1145].IN:= (GTAC_CONFIG.Option_Robot_Count>=25) AND
							(MAIN.R25.Battery_Alarm OR (MAIN.R25.Faulted AND MAIN.Control_Power_ON));
		Out_To_ICxx.System_Faults[1145]:=Fault_Tmrs[1145].Q;
	(*Fault1146 - R26 System Fault*)
		Fault_Tmrs[1146].PT:=Short_Faults;
		Fault_Tmrs[1146]();
		Fault_Tmrs[1146].IN:= (GTAC_CONFIG.Option_Robot_Count>=26) AND
							(MAIN.R26.Battery_Alarm OR (MAIN.R26.Faulted AND MAIN.Control_Power_ON));
		Out_To_ICxx.System_Faults[1146]:=Fault_Tmrs[1146].Q;
	(*Fault1147 - R27 System Fault*)
		Fault_Tmrs[1147].PT:=Short_Faults;
		Fault_Tmrs[1147]();
		Fault_Tmrs[1147].IN:= (GTAC_CONFIG.Option_Robot_Count>=27) AND
							(MAIN.R27.Battery_Alarm OR (MAIN.R27.Faulted AND MAIN.Control_Power_ON));
		Out_To_ICxx.System_Faults[1147]:=Fault_Tmrs[1147].Q;
	(*Fault1148 - R28 System Fault*)
		Fault_Tmrs[1148].PT:=Short_Faults;
		Fault_Tmrs[1148]();
		Fault_Tmrs[1148].IN:= (GTAC_CONFIG.Option_Robot_Count>=28) AND
							(MAIN.R28.Battery_Alarm OR (MAIN.R28.Faulted AND MAIN.Control_Power_ON));
		Out_To_ICxx.System_Faults[1148]:=Fault_Tmrs[1148].Q;
	(*Fault1149 - R29 System Fault*)
		Fault_Tmrs[1149].PT:=Short_Faults;
		Fault_Tmrs[1149]();
		Fault_Tmrs[1149].IN:= (GTAC_CONFIG.Option_Robot_Count>=29) AND
							(MAIN.R29.Battery_Alarm OR (MAIN.R29.Faulted AND MAIN.Control_Power_ON));
		Out_To_ICxx.System_Faults[1149]:=Fault_Tmrs[1149].Q;
	(*Fault1150 - R30 System Fault*)
		Fault_Tmrs[1150].PT:=Short_Faults;
		Fault_Tmrs[1150]();
		Fault_Tmrs[1150].IN:= (GTAC_CONFIG.Option_Robot_Count>=30) AND
							(MAIN.R30.Battery_Alarm OR (MAIN.R30.Faulted AND MAIN.Control_Power_ON));
		Out_To_ICxx.System_Faults[1150]:=Fault_Tmrs[1150].Q;

	(*------------------------------------------------------------------------------------------- Robot TQM (Torque Monitoring) Not Valid Faults ---------------------------------------------------------------------------*)
	(*Fault1151 - R1 TQM Not Valid*)
		Fault_Tmrs[1151].PT:=Short_Faults;
		Fault_Tmrs[1151]();
		Fault_Tmrs[1151].IN:= (GTAC_CONFIG.Option_Robot_Count>=1)  AND
							MAIN.R1.TQM_NotValid_FLT;
		Out_To_ICxx.System_Faults[1151]:=Fault_Tmrs[1151].Q;
	(*Fault1152 - R2 TQM Not Valid*)
		Fault_Tmrs[1152].PT:=Short_Faults;
		Fault_Tmrs[1152]();
		Fault_Tmrs[1152].IN:= (GTAC_CONFIG.Option_Robot_Count>=2)  AND
							MAIN.R2.TQM_NotValid_FLT;
		Out_To_ICxx.System_Faults[1152]:=Fault_Tmrs[1152].Q;
	(*Fault1153 - R3 TQM Not Valid*)
		Fault_Tmrs[1153].PT:=Short_Faults;
		Fault_Tmrs[1153]();
		Fault_Tmrs[1153].IN:= (GTAC_CONFIG.Option_Robot_Count>=3)  AND
							MAIN.R3.TQM_NotValid_FLT;
		Out_To_ICxx.System_Faults[1153]:=Fault_Tmrs[1153].Q;
	(*Fault1154 - R4 TQM Not Valid*)
		Fault_Tmrs[1154].PT:=Short_Faults;
		Fault_Tmrs[1154]();
		Fault_Tmrs[1154].IN:=(GTAC_CONFIG.Option_Robot_Count>=4)  AND
							MAIN.R4.TQM_NotValid_FLT;
		Out_To_ICxx.System_Faults[1154]:=Fault_Tmrs[1154].Q;
	(*Fault1155 - R5 TQM Not Valid*)
		Fault_Tmrs[1155].PT:=Short_Faults;
		Fault_Tmrs[1155]();
		Fault_Tmrs[1155].IN:= (GTAC_CONFIG.Option_Robot_Count>=5)  AND
							MAIN.R5.TQM_NotValid_FLT;
		Out_To_ICxx.System_Faults[1155]:=Fault_Tmrs[1155].Q;
	(*Fault1156 - R6 TQM Not Valid*)
		Fault_Tmrs[1156].PT:=Short_Faults;
		Fault_Tmrs[1156]();
		Fault_Tmrs[1156].IN:= (GTAC_CONFIG.Option_Robot_Count>=6)  AND
							MAIN.R6.TQM_NotValid_FLT;
		Out_To_ICxx.System_Faults[1156]:=Fault_Tmrs[1156].Q;
	(*Fault1157 - R10 TQM Not Valid*)
		Fault_Tmrs[1157].PT:=Short_Faults;
		Fault_Tmrs[1157]();
		Fault_Tmrs[1157].IN:= (GTAC_CONFIG.Option_Robot_Count>=7)  AND
							MAIN.R7.TQM_NotValid_FLT;
		Out_To_ICxx.System_Faults[1157]:=Fault_Tmrs[1157].Q;
	(*Fault1158 - R8 TQM Not Valid*)
		Fault_Tmrs[1158].PT:=Short_Faults;
		Fault_Tmrs[1158]();
		Fault_Tmrs[1158].IN:= (GTAC_CONFIG.Option_Robot_Count>=8)  AND
							MAIN.R8.TQM_NotValid_FLT;
		Out_To_ICxx.System_Faults[1158]:=Fault_Tmrs[1158].Q;
	(*Fault1159 - R9 TQM Not Valid*)
		Fault_Tmrs[1159].PT:=Short_Faults;
		Fault_Tmrs[1159]();
		Fault_Tmrs[1159].IN:= (GTAC_CONFIG.Option_Robot_Count>=9)  AND
							MAIN.R9.TQM_NotValid_FLT;
		Out_To_ICxx.System_Faults[1159]:=Fault_Tmrs[1159].Q;
	(*Fault1160 - R10 TQM Not Valid*)
		Fault_Tmrs[1160].PT:=Short_Faults;
		Fault_Tmrs[1160]();
		Fault_Tmrs[1160].IN:= (GTAC_CONFIG.Option_Robot_Count>=10)  AND
							MAIN.R10.TQM_NotValid_FLT;
		Out_To_ICxx.System_Faults[1160]:=Fault_Tmrs[1160].Q;
	(*Fault1161 - R11 TQM Not Valid*)
		Fault_Tmrs[1161].PT:=Short_Faults;
		Fault_Tmrs[1161]();
		Fault_Tmrs[1161].IN:= (GTAC_CONFIG.Option_Robot_Count>=11)  AND
							MAIN.R11.TQM_NotValid_FLT;
		Out_To_ICxx.System_Faults[1161]:=Fault_Tmrs[1161].Q;
	(*Fault1162 - R12 TQM Not Valid*)
		Fault_Tmrs[1162].PT:=Short_Faults;
		Fault_Tmrs[1162]();
		Fault_Tmrs[1162].IN:= (GTAC_CONFIG.Option_Robot_Count>=12)  AND
							MAIN.R12.TQM_NotValid_FLT;
		Out_To_ICxx.System_Faults[1162]:=Fault_Tmrs[1162].Q;
	(*Fault1163 - R13 TQM Not Valid*)
		Fault_Tmrs[1163].PT:=Short_Faults;
		Fault_Tmrs[1163]();
		Fault_Tmrs[1163].IN:= (GTAC_CONFIG.Option_Robot_Count>=13)  AND
							MAIN.R13.TQM_NotValid_FLT;
		Out_To_ICxx.System_Faults[1163]:=Fault_Tmrs[1163].Q;
	(*Fault1164 - R14 TQM Not Valid*)
		Fault_Tmrs[1164].PT:=Short_Faults;
		Fault_Tmrs[1164]();
		Fault_Tmrs[1164].IN:= (GTAC_CONFIG.Option_Robot_Count>=14)  AND
							MAIN.R14.TQM_NotValid_FLT;
		Out_To_ICxx.System_Faults[1164]:=Fault_Tmrs[1164].Q;
	(*Fault1165 - R15 TQM Not Valid*)
		Fault_Tmrs[1165].PT:=Short_Faults;
		Fault_Tmrs[1165]();
		Fault_Tmrs[1165].IN:= (GTAC_CONFIG.Option_Robot_Count>=15)  AND
							MAIN.R15.TQM_NotValid_FLT;
		Out_To_ICxx.System_Faults[1165]:=Fault_Tmrs[1165].Q;
	(*Fault1166 - R16 TQM Not Valid*)
		Fault_Tmrs[1166].PT:=Short_Faults;
		Fault_Tmrs[1166]();
		Fault_Tmrs[1166].IN:= (GTAC_CONFIG.Option_Robot_Count>=16)  AND
							MAIN.R16.TQM_NotValid_FLT;
		Out_To_ICxx.System_Faults[1166]:=Fault_Tmrs[1166].Q;
	(*Fault1167 - R17 TQM Not Valid*)
		Fault_Tmrs[1167].PT:=Short_Faults;
		Fault_Tmrs[1167]();
		Fault_Tmrs[1167].IN:= (GTAC_CONFIG.Option_Robot_Count>=17)  AND
							MAIN.R17.TQM_NotValid_FLT;
		Out_To_ICxx.System_Faults[1167]:=Fault_Tmrs[1167].Q;
	(*Fault1168 - R18 TQM Not Valid*)
		Fault_Tmrs[1168].PT:=Short_Faults;
		Fault_Tmrs[1168]();
		Fault_Tmrs[1168].IN:= (GTAC_CONFIG.Option_Robot_Count>=18)  AND
							MAIN.R18.TQM_NotValid_FLT;
		Out_To_ICxx.System_Faults[1168]:=Fault_Tmrs[1168].Q;
	(*Fault1169 - R19 TQM Not Valid*)
		Fault_Tmrs[1169].PT:=Short_Faults;
		Fault_Tmrs[1169]();
		Fault_Tmrs[1169].IN:= (GTAC_CONFIG.Option_Robot_Count>=19)  AND
							MAIN.R19.TQM_NotValid_FLT;
		Out_To_ICxx.System_Faults[1169]:=Fault_Tmrs[1169].Q;
	(*Fault1170 - R20 TQM Not Valid*)
		Fault_Tmrs[1170].PT:=Short_Faults;
		Fault_Tmrs[1170]();
		Fault_Tmrs[1170].IN:= (GTAC_CONFIG.Option_Robot_Count>=20)  AND
							MAIN.R20.TQM_NotValid_FLT;
		Out_To_ICxx.System_Faults[1170]:=Fault_Tmrs[1170].Q;
	(*Fault1171 - R21 TQM Not Valid*)
		Fault_Tmrs[1171].PT:=Short_Faults;
		Fault_Tmrs[1171]();
		Fault_Tmrs[1171].IN:= (GTAC_CONFIG.Option_Robot_Count>=21)  AND
							MAIN.R21.TQM_NotValid_FLT;
		Out_To_ICxx.System_Faults[1171]:=Fault_Tmrs[1171].Q;
	(*Fault1172 - R22 TQM Not Valid*)
		Fault_Tmrs[1172].PT:=Short_Faults;
		Fault_Tmrs[1172]();
		Fault_Tmrs[1172].IN:= (GTAC_CONFIG.Option_Robot_Count>=22)  AND
							MAIN.R22.TQM_NotValid_FLT;
		Out_To_ICxx.System_Faults[1172]:=Fault_Tmrs[1172].Q;
	(*Fault1173 - R23 TQM Not Valid*)
		Fault_Tmrs[1173].PT:=Short_Faults;
		Fault_Tmrs[1173]();
		Fault_Tmrs[1173].IN:= (GTAC_CONFIG.Option_Robot_Count>=23)  AND
							MAIN.R23.TQM_NotValid_FLT;
		Out_To_ICxx.System_Faults[1173]:=Fault_Tmrs[1173].Q;
	(*Fault1174 - R24 TQM Not Valid*)
		Fault_Tmrs[1174].PT:=Short_Faults;
		Fault_Tmrs[1174]();
		Fault_Tmrs[1174].IN:= (GTAC_CONFIG.Option_Robot_Count>=24)  AND
							MAIN.R24.TQM_NotValid_FLT;
		Out_To_ICxx.System_Faults[1174]:=Fault_Tmrs[1174].Q;
	(*Fault1175 - R25 TQM Not Valid*)
		Fault_Tmrs[1175].PT:=Short_Faults;
		Fault_Tmrs[1175]();
		Fault_Tmrs[1175].IN:= (GTAC_CONFIG.Option_Robot_Count>=25)  AND
							MAIN.R25.TQM_NotValid_FLT;
		Out_To_ICxx.System_Faults[1175]:=Fault_Tmrs[1175].Q;
	(*Fault1176 - R26 TQM Not Valid*)
		Fault_Tmrs[1176].PT:=Short_Faults;
		Fault_Tmrs[1176]();
		Fault_Tmrs[1176].IN:= (GTAC_CONFIG.Option_Robot_Count>=26)  AND
							MAIN.R26.TQM_NotValid_FLT;
		Out_To_ICxx.System_Faults[1176]:=Fault_Tmrs[1176].Q;
	(*Fault1177 - R27 TQM Not Valid*)
		Fault_Tmrs[1177].PT:=Short_Faults;
		Fault_Tmrs[1177]();
		Fault_Tmrs[1177].IN:= (GTAC_CONFIG.Option_Robot_Count>=27)  AND
							MAIN.R27.TQM_NotValid_FLT;
		Out_To_ICxx.System_Faults[1177]:=Fault_Tmrs[1177].Q;
	(*Fault1178 - R28 TQM Not Valid*)
		Fault_Tmrs[1178].PT:=Short_Faults;
		Fault_Tmrs[1178]();
		Fault_Tmrs[1178].IN:= (GTAC_CONFIG.Option_Robot_Count>=28)  AND
							MAIN.R28.TQM_NotValid_FLT;
		Out_To_ICxx.System_Faults[1178]:=Fault_Tmrs[1178].Q;
	(*Fault1179 - R29 TQM Not Valid*)
		Fault_Tmrs[1179].PT:=Short_Faults;
		Fault_Tmrs[1179]();
		Fault_Tmrs[1179].IN:= (GTAC_CONFIG.Option_Robot_Count>=29)  AND
							MAIN.R29.TQM_NotValid_FLT;
		Out_To_ICxx.System_Faults[1179]:=Fault_Tmrs[1179].Q;
	(*Fault1180 - R30 TQM Not Valid*)
		Fault_Tmrs[1180].PT:=Short_Faults;
		Fault_Tmrs[1180]();
		Fault_Tmrs[1180].IN:= (GTAC_CONFIG.Option_Robot_Count>=30)  AND
							MAIN.R30.TQM_NotValid_FLT;
		Out_To_ICxx.System_Faults[1180]:=Fault_Tmrs[1180].Q;

	(*-------------------------------------------------------------------------------- Robot SafeOP Active Faults -------------------------------------------------------------------*)
	(*Fault1181 - R1 SafeOP Not Active Fault*)
		Fault_Tmrs[1181].PT:= Short_Faults;
		Fault_Tmrs[1181]();
		Fault_Tmrs[1181].IN:= (GTAC_CONFIG.Option_Robot_Count>=1)  AND
							NOT MAIN.R1.SafeOP_Active AND (MAIN.R1.FB_In.Robot_Type >=61);
		Out_To_ICxx.System_Faults[1181]:=Fault_Tmrs[1181].Q;
	(*Fault1182 - R2 SafeOP Not Active Fault*)
		Fault_Tmrs[1182].PT:= Short_Faults;
		Fault_Tmrs[1182]();
		Fault_Tmrs[1182].IN:= (GTAC_CONFIG.Option_Robot_Count>=2)  AND
							NOT MAIN.R2.SafeOP_Active AND (MAIN.R2.FB_In.Robot_Type >=61);
		Out_To_ICxx.System_Faults[1182]:=Fault_Tmrs[1182].Q;
	(*Fault1183 - R3 SafeOP Not Active Fault*)
		Fault_Tmrs[1183].PT:= Short_Faults;
		Fault_Tmrs[1183]();
		Fault_Tmrs[1183].IN:= (GTAC_CONFIG.Option_Robot_Count>=3)  AND
							NOT MAIN.R3.SafeOP_Active AND (MAIN.R3.FB_In.Robot_Type >=61);
		Out_To_ICxx.System_Faults[1183]:=Fault_Tmrs[1183].Q;
	(*Fault1184 - R4 SafeOP Not Active Fault*)
		Fault_Tmrs[1184].PT:= Short_Faults;
		Fault_Tmrs[1184]();
		Fault_Tmrs[1184].IN:= (GTAC_CONFIG.Option_Robot_Count>=4)  AND
							NOT MAIN.R4.SafeOP_Active AND (MAIN.R4.FB_In.Robot_Type >=61);
		Out_To_ICxx.System_Faults[1184]:=Fault_Tmrs[1184].Q;
	(*Fault1185 - R5 SafeOP Not Active Fault*)
		Fault_Tmrs[1185].PT:= Short_Faults;
		Fault_Tmrs[1185]();
		Fault_Tmrs[1185].IN:= (GTAC_CONFIG.Option_Robot_Count>=5)  AND
							NOT MAIN.R5.SafeOP_Active AND (MAIN.R5.FB_In.Robot_Type >=61);
		Out_To_ICxx.System_Faults[1185]:=Fault_Tmrs[1185].Q;
	(*Fault1186 - R6 SafeOP Not Active Fault*)
		Fault_Tmrs[1186].PT:= Short_Faults;
		Fault_Tmrs[1186]();
		Fault_Tmrs[1186].IN:= (GTAC_CONFIG.Option_Robot_Count>=6)  AND
							NOT MAIN.R6.SafeOP_Active AND (MAIN.R6.FB_In.Robot_Type >=61);
		Out_To_ICxx.System_Faults[1186]:=Fault_Tmrs[1186].Q;
	(*Fault1187 - R7 SafeOP Not Active Fault*)
		Fault_Tmrs[1187].PT:= Short_Faults;
		Fault_Tmrs[1187]();
		Fault_Tmrs[1187].IN:= (GTAC_CONFIG.Option_Robot_Count>=7)  AND
							NOT MAIN.R7.SafeOP_Active AND (MAIN.R7.FB_In.Robot_Type >=61);
		Out_To_ICxx.System_Faults[1187]:=Fault_Tmrs[1187].Q;
	(*Fault1188 - R8 SafeOP Not Active Fault*)
		Fault_Tmrs[1188].PT:= Short_Faults;
		Fault_Tmrs[1188]();
		Fault_Tmrs[1188].IN:= (GTAC_CONFIG.Option_Robot_Count>=8)  AND
							NOT MAIN.R8.SafeOP_Active AND (MAIN.R8.FB_In.Robot_Type >=61);
		Out_To_ICxx.System_Faults[1188]:=Fault_Tmrs[1188].Q;
	(*Fault1189 - R9 SafeOP Not Active Fault*)
		Fault_Tmrs[1189].PT:= Short_Faults;
		Fault_Tmrs[1189]();
		Fault_Tmrs[1189].IN:= (GTAC_CONFIG.Option_Robot_Count>=9)  AND
							NOT MAIN.R9.SafeOP_Active AND (MAIN.R9.FB_In.Robot_Type >=61);
		Out_To_ICxx.System_Faults[1189]:=Fault_Tmrs[1189].Q;
	(*Fault1190 - R10 SafeOP Not Active Fault*)
		Fault_Tmrs[1190].PT:= Short_Faults;
		Fault_Tmrs[1190]();
		Fault_Tmrs[1190].IN:= (GTAC_CONFIG.Option_Robot_Count>=10)  AND
							NOT MAIN.R10.SafeOP_Active AND (MAIN.R10.FB_In.Robot_Type >=61);
		Out_To_ICxx.System_Faults[1190]:=Fault_Tmrs[1190].Q;
	(*Fault1191 - R11 SafeOP Not Active Fault*)
		Fault_Tmrs[1191].PT:= Short_Faults;
		Fault_Tmrs[1191]();
		Fault_Tmrs[1191].IN:= (GTAC_CONFIG.Option_Robot_Count>=11)  AND
							NOT MAIN.R11.SafeOP_Active AND (MAIN.R11.FB_In.Robot_Type >=61);
		Out_To_ICxx.System_Faults[1191]:=Fault_Tmrs[1191].Q;
	(*Fault1192 - R12 SafeOP Not Active Fault*)
		Fault_Tmrs[1192].PT:= Short_Faults;
		Fault_Tmrs[1192]();
		Fault_Tmrs[1192].IN:= (GTAC_CONFIG.Option_Robot_Count>=12)  AND
							NOT MAIN.R12.SafeOP_Active AND (MAIN.R12.FB_In.Robot_Type >=61);
		Out_To_ICxx.System_Faults[1192]:=Fault_Tmrs[1192].Q;
	(*Fault1193 - R13 SafeOP Not Active Fault*)
		Fault_Tmrs[1193].PT:= Short_Faults;
		Fault_Tmrs[1193]();
		Fault_Tmrs[1193].IN:= (GTAC_CONFIG.Option_Robot_Count>=13)  AND
							NOT MAIN.R13.SafeOP_Active AND (MAIN.R13.FB_In.Robot_Type >=61);
		Out_To_ICxx.System_Faults[1193]:=Fault_Tmrs[1193].Q;
	(*Fault1194 - R14 SafeOP Not Active Fault*)
		Fault_Tmrs[1194].PT:= Short_Faults;
		Fault_Tmrs[1194]();
		Fault_Tmrs[1194].IN:= (GTAC_CONFIG.Option_Robot_Count>=14)  AND
							NOT MAIN.R14.SafeOP_Active AND (MAIN.R14.FB_In.Robot_Type >=61);
		Out_To_ICxx.System_Faults[1194]:=Fault_Tmrs[1194].Q;
	(*Fault1195 - R15 SafeOP Not Active Fault*)
		Fault_Tmrs[1195].PT:= Short_Faults;
		Fault_Tmrs[1195]();
		Fault_Tmrs[1195].IN:= (GTAC_CONFIG.Option_Robot_Count>=15)  AND
							NOT MAIN.R15.SafeOP_Active AND (MAIN.R15.FB_In.Robot_Type >=61);
		Out_To_ICxx.System_Faults[1195]:=Fault_Tmrs[1195].Q;
	(*Fault1196 - R16 SafeOP Not Active Fault*)
		Fault_Tmrs[1196].PT:= Short_Faults;
		Fault_Tmrs[1196]();
		Fault_Tmrs[1196].IN:= (GTAC_CONFIG.Option_Robot_Count>=16)  AND
							NOT MAIN.R16.SafeOP_Active AND (MAIN.R16.FB_In.Robot_Type >=61);
		Out_To_ICxx.System_Faults[1196]:=Fault_Tmrs[1196].Q;
	(*Fault1197 - R17 SafeOP Not Active Fault*)
		Fault_Tmrs[1197].PT:= Short_Faults;
		Fault_Tmrs[1197]();
		Fault_Tmrs[1197].IN:= (GTAC_CONFIG.Option_Robot_Count>=17)  AND
							NOT MAIN.R17.SafeOP_Active AND (MAIN.R17.FB_In.Robot_Type >=61);
		Out_To_ICxx.System_Faults[1197]:=Fault_Tmrs[1197].Q;
	(*Fault1198 - R18 SafeOP Not Active Fault*)
		Fault_Tmrs[1198].PT:= Short_Faults;
		Fault_Tmrs[1198]();
		Fault_Tmrs[1198].IN:= (GTAC_CONFIG.Option_Robot_Count>=18)  AND
							NOT MAIN.R18.SafeOP_Active AND (MAIN.R18.FB_In.Robot_Type >=61);
		Out_To_ICxx.System_Faults[1198]:=Fault_Tmrs[1198].Q;
	(*Fault1199 - R19 SafeOP Not Active Fault*)
		Fault_Tmrs[1199].PT:= Short_Faults;
		Fault_Tmrs[1199]();
		Fault_Tmrs[1199].IN:= (GTAC_CONFIG.Option_Robot_Count>=19)  AND
							NOT MAIN.R19.SafeOP_Active AND (MAIN.R19.FB_In.Robot_Type >=61);
		Out_To_ICxx.System_Faults[1199]:=Fault_Tmrs[1199].Q;
	(*Fault1200 - R20 SafeOP Not Active Fault*)
		Fault_Tmrs[1200].PT:= Short_Faults;
		Fault_Tmrs[1200]();
		Fault_Tmrs[1200].IN:= (GTAC_CONFIG.Option_Robot_Count>=20)  AND
							NOT MAIN.R20.SafeOP_Active AND (MAIN.R20.FB_In.Robot_Type >=61);
		Out_To_ICxx.System_Faults[1200]:=Fault_Tmrs[1200].Q;
	(*Fault1201 - R21 SafeOP Not Active Fault*)
		Fault_Tmrs[1201].PT:= Short_Faults;
		Fault_Tmrs[1201]();
		Fault_Tmrs[1201].IN:= (GTAC_CONFIG.Option_Robot_Count>=21)  AND
							NOT MAIN.R21.SafeOP_Active AND (MAIN.R21.FB_In.Robot_Type >=61);
		Out_To_ICxx.System_Faults[1201]:=Fault_Tmrs[1201].Q;
	(*Fault1202 - R22 SafeOP Not Active Fault*)
		Fault_Tmrs[1202].PT:= Short_Faults;
		Fault_Tmrs[1202]();
		Fault_Tmrs[1202].IN:= (GTAC_CONFIG.Option_Robot_Count>=22)  AND
							NOT MAIN.R22.SafeOP_Active AND (MAIN.R22.FB_In.Robot_Type >=61);
		Out_To_ICxx.System_Faults[1202]:=Fault_Tmrs[1202].Q;
	(*Fault1203 - R23 SafeOP Not Active Fault*)
		Fault_Tmrs[1203].PT:= Short_Faults;
		Fault_Tmrs[1203]();
		Fault_Tmrs[1203].IN:= (GTAC_CONFIG.Option_Robot_Count>=23)  AND
							NOT MAIN.R23.SafeOP_Active AND (MAIN.R23.FB_In.Robot_Type >=61);
		Out_To_ICxx.System_Faults[1203]:=Fault_Tmrs[1203].Q;
	(*Fault1204 - R24 SafeOP Not Active Fault*)
		Fault_Tmrs[1204].PT:= Short_Faults;
		Fault_Tmrs[1204]();
		Fault_Tmrs[1204].IN:= (GTAC_CONFIG.Option_Robot_Count>=24)  AND
							NOT MAIN.R24.SafeOP_Active AND (MAIN.R24.FB_In.Robot_Type >=61);
		Out_To_ICxx.System_Faults[1204]:=Fault_Tmrs[1204].Q;
	(*Fault1205 - R25 SafeOP Not Active Fault*)
		Fault_Tmrs[1205].PT:= Short_Faults;
		Fault_Tmrs[1205]();
		Fault_Tmrs[1205].IN:= (GTAC_CONFIG.Option_Robot_Count>=25)  AND
							NOT MAIN.R25.SafeOP_Active AND (MAIN.R25.FB_In.Robot_Type >=61);
		Out_To_ICxx.System_Faults[1205]:=Fault_Tmrs[1205].Q;
	(*Fault1206 - R26 SafeOP Not Active Fault*)
		Fault_Tmrs[1206].PT:= Short_Faults;
		Fault_Tmrs[1206]();
		Fault_Tmrs[1206].IN:= (GTAC_CONFIG.Option_Robot_Count>=26)  AND
							NOT MAIN.R26.SafeOP_Active AND (MAIN.R26.FB_In.Robot_Type >=61);
		Out_To_ICxx.System_Faults[1206]:=Fault_Tmrs[1206].Q;
	(*Fault1207 - R27 SafeOP Not Active Fault*)
		Fault_Tmrs[1207].PT:= Short_Faults;
		Fault_Tmrs[1207]();
		Fault_Tmrs[1207].IN:= (GTAC_CONFIG.Option_Robot_Count>=27)  AND
							NOT MAIN.R27.SafeOP_Active AND (MAIN.R27.FB_In.Robot_Type >=61);
		Out_To_ICxx.System_Faults[1207]:=Fault_Tmrs[1207].Q;
	(*Fault1208 - R28 SafeOP Not Active Fault*)
		Fault_Tmrs[1208].PT:= Short_Faults;
		Fault_Tmrs[1208]();
		Fault_Tmrs[1208].IN:= (GTAC_CONFIG.Option_Robot_Count>=28)  AND
							NOT MAIN.R28.SafeOP_Active AND (MAIN.R28.FB_In.Robot_Type >=61);
		Out_To_ICxx.System_Faults[1208]:=Fault_Tmrs[1208].Q;
	(*Fault1209 - R29 SafeOP Not Active Fault*)
		Fault_Tmrs[1209].PT:= Short_Faults;
		Fault_Tmrs[1209]();
		Fault_Tmrs[1209].IN:= (GTAC_CONFIG.Option_Robot_Count>=29)  AND
							NOT MAIN.R29.SafeOP_Active AND (MAIN.R29.FB_In.Robot_Type >=61);
		Out_To_ICxx.System_Faults[1209]:=Fault_Tmrs[1209].Q;
	(*Fault1210 - R30 SafeOP Not Active Fault*)
		Fault_Tmrs[1210].PT:= Short_Faults;
		Fault_Tmrs[1210]();
		Fault_Tmrs[1210].IN:= (GTAC_CONFIG.Option_Robot_Count>=30)  AND
							NOT MAIN.R30.SafeOP_Active AND (MAIN.R30.FB_In.Robot_Type >=61);
		Out_To_ICxx.System_Faults[1210]:=Fault_Tmrs[1210].Q;

	(* --------------------------------------------------------------------- Robot Ack ID Faults -------------------------------------------------------------------------------*)
	(*Fault1211 - R1 Ack ID Fault*)
		Fault_Tmrs[1211].PT:= Short_Faults;
		Fault_Tmrs[1211]();
		Fault_Tmrs[1211].IN:= (GTAC_CONFIG.Option_Robot_Count>=1) AND
							MAIN.R1.Ack_ID_FLT;
		Out_To_ICxx.System_Faults[1211]:=Fault_Tmrs[1211].Q;
	(*Fault1212 - R2 Ack ID Fault*)
		Fault_Tmrs[1212].PT:= Short_Faults;
		Fault_Tmrs[1212]();
		Fault_Tmrs[1212].IN:= (GTAC_CONFIG.Option_Robot_Count>=2) AND
							MAIN.R2.Ack_ID_FLT;
		Out_To_ICxx.System_Faults[1212]:=Fault_Tmrs[1212].Q;
	(*Fault1213 - R3 Ack ID Fault*)
		Fault_Tmrs[1213].PT:= Short_Faults;
		Fault_Tmrs[1213]();
		Fault_Tmrs[1213].IN:= (GTAC_CONFIG.Option_Robot_Count>=3) AND
							MAIN.R3.Ack_ID_FLT;
		Out_To_ICxx.System_Faults[1213]:=Fault_Tmrs[1213].Q;
	(*Fault1214 - R4 Ack ID Fault*)
		Fault_Tmrs[1214].PT:= Short_Faults;
		Fault_Tmrs[1214]();
		Fault_Tmrs[1214].IN:= (GTAC_CONFIG.Option_Robot_Count>=4) AND
							MAIN.R4.Ack_ID_FLT;
		Out_To_ICxx.System_Faults[1214]:=Fault_Tmrs[1214].Q;
	(*Fault1215 - R5 Ack ID Fault*)
		Fault_Tmrs[1215].PT:= Short_Faults;
		Fault_Tmrs[1215]();
		Fault_Tmrs[1215].IN:= (GTAC_CONFIG.Option_Robot_Count>=5) AND
							MAIN.R5.Ack_ID_FLT;
		Out_To_ICxx.System_Faults[1215]:=Fault_Tmrs[1215].Q;
	(*Fault1216 - R6 Ack ID Fault*)
		Fault_Tmrs[1216].PT:= Short_Faults;
		Fault_Tmrs[1216]();
		Fault_Tmrs[1216].IN:= (GTAC_CONFIG.Option_Robot_Count>=6) AND
							MAIN.R6.Ack_ID_FLT;
		Out_To_ICxx.System_Faults[1216]:=Fault_Tmrs[1216].Q;
	(*Fault1217 - R7 Ack ID Fault*)
		Fault_Tmrs[1217].PT:= Short_Faults;
		Fault_Tmrs[1217]();
		Fault_Tmrs[1217].IN:= (GTAC_CONFIG.Option_Robot_Count>=7) AND
							MAIN.R7.Ack_ID_FLT;
		Out_To_ICxx.System_Faults[1217]:=Fault_Tmrs[1217].Q;
	(*Fault1218 - R8 Ack ID Fault*)
		Fault_Tmrs[1218].PT:= Short_Faults;
		Fault_Tmrs[1218]();
		Fault_Tmrs[1218].IN:= (GTAC_CONFIG.Option_Robot_Count>=8) AND
							MAIN.R8.Ack_ID_FLT;
		Out_To_ICxx.System_Faults[1218]:=Fault_Tmrs[1218].Q;
	(*Fault1219 - R9 Ack ID Fault*)
		Fault_Tmrs[1219].PT:= Short_Faults;
		Fault_Tmrs[1219]();
		Fault_Tmrs[1219].IN:= (GTAC_CONFIG.Option_Robot_Count>=9) AND
							MAIN.R9.Ack_ID_FLT;
		Out_To_ICxx.System_Faults[1219]:=Fault_Tmrs[1219].Q;
	(*Fault1220 - R10 Ack ID Fault*)
		Fault_Tmrs[1220].PT:= Short_Faults;
		Fault_Tmrs[1220]();
		Fault_Tmrs[1220].IN:= (GTAC_CONFIG.Option_Robot_Count>=10) AND
							MAIN.R10.Ack_ID_FLT;
		Out_To_ICxx.System_Faults[1220]:=Fault_Tmrs[1220].Q;
	(*Fault1221 - R11 Ack ID Fault*)
		Fault_Tmrs[1221].PT:= Short_Faults;
		Fault_Tmrs[1221]();
		Fault_Tmrs[1221].IN:= (GTAC_CONFIG.Option_Robot_Count>=11) AND
							MAIN.R11.Ack_ID_FLT;
		Out_To_ICxx.System_Faults[1221]:=Fault_Tmrs[1221].Q;
	(*Fault1222 - R12 Ack ID Fault*)
		Fault_Tmrs[1222].PT:= Short_Faults;
		Fault_Tmrs[1222]();
		Fault_Tmrs[1222].IN:= (GTAC_CONFIG.Option_Robot_Count>=12) AND
							MAIN.R12.Ack_ID_FLT;
		Out_To_ICxx.System_Faults[1222]:=Fault_Tmrs[1222].Q;
	(*Fault1223 - R13 Ack ID Fault*)
		Fault_Tmrs[1223].PT:= Short_Faults;
		Fault_Tmrs[1223]();
		Fault_Tmrs[1223].IN:= (GTAC_CONFIG.Option_Robot_Count>=13) AND
							MAIN.R13.Ack_ID_FLT;
		Out_To_ICxx.System_Faults[1223]:=Fault_Tmrs[1223].Q;
	(*Fault1224 - R14 Ack ID Fault*)
		Fault_Tmrs[1224].PT:= Short_Faults;
		Fault_Tmrs[1224]();
		Fault_Tmrs[1224].IN:= (GTAC_CONFIG.Option_Robot_Count>=14) AND
							MAIN.R14.Ack_ID_FLT;
		Out_To_ICxx.System_Faults[1224]:=Fault_Tmrs[1224].Q;
	(*Fault1225 - R15 Ack ID Fault*)
		Fault_Tmrs[1225].PT:= Short_Faults;
		Fault_Tmrs[1225]();
		Fault_Tmrs[1225].IN:= (GTAC_CONFIG.Option_Robot_Count>=15) AND
							MAIN.R15.Ack_ID_FLT;
		Out_To_ICxx.System_Faults[1225]:=Fault_Tmrs[1225].Q;
	(*Fault1226 - R16 Ack ID Fault*)
		Fault_Tmrs[1226].PT:= Short_Faults;
		Fault_Tmrs[1226]();
		Fault_Tmrs[1226].IN:= (GTAC_CONFIG.Option_Robot_Count>=16) AND
							MAIN.R16.Ack_ID_FLT;
		Out_To_ICxx.System_Faults[1226]:=Fault_Tmrs[1226].Q;
	(*Fault1227 - R17 Ack ID Fault*)
		Fault_Tmrs[1227].PT:= Short_Faults;
		Fault_Tmrs[1227]();
		Fault_Tmrs[1227].IN:= (GTAC_CONFIG.Option_Robot_Count>=17) AND
							MAIN.R17.Ack_ID_FLT;
		Out_To_ICxx.System_Faults[1227]:=Fault_Tmrs[1227].Q;
	(*Fault1228 - R18 Ack ID Fault*)
		Fault_Tmrs[1228].PT:= Short_Faults;
		Fault_Tmrs[1228]();
		Fault_Tmrs[1228].IN:= (GTAC_CONFIG.Option_Robot_Count>=18) AND
							MAIN.R18.Ack_ID_FLT;
		Out_To_ICxx.System_Faults[1228]:=Fault_Tmrs[1228].Q;
	(*Fault1229 - R19 Ack ID Fault*)
		Fault_Tmrs[1229].PT:= Short_Faults;
		Fault_Tmrs[1229]();
		Fault_Tmrs[1229].IN:= (GTAC_CONFIG.Option_Robot_Count>=19) AND
							MAIN.R19.Ack_ID_FLT;
		Out_To_ICxx.System_Faults[1229]:=Fault_Tmrs[1229].Q;
	(*Fault1230 - R20 Ack ID Fault*)
		Fault_Tmrs[1230].PT:= Short_Faults;
		Fault_Tmrs[1230]();
		Fault_Tmrs[1230].IN:= (GTAC_CONFIG.Option_Robot_Count>=20) AND
							MAIN.R20.Ack_ID_FLT;
		Out_To_ICxx.System_Faults[1230]:=Fault_Tmrs[1230].Q;
	(*Fault1231 - R21 Ack ID Fault*)
		Fault_Tmrs[1231].PT:= Short_Faults;
		Fault_Tmrs[1231]();
		Fault_Tmrs[1231].IN:= (GTAC_CONFIG.Option_Robot_Count>=21) AND
							MAIN.R21.Ack_ID_FLT;
		Out_To_ICxx.System_Faults[1231]:=Fault_Tmrs[1231].Q;
	(*Fault1232 - R22 Ack ID Fault*)
		Fault_Tmrs[1232].PT:= Short_Faults;
		Fault_Tmrs[1232]();
		Fault_Tmrs[1232].IN:= (GTAC_CONFIG.Option_Robot_Count>=22) AND
							MAIN.R22.Ack_ID_FLT;
		Out_To_ICxx.System_Faults[1232]:=Fault_Tmrs[1232].Q;
	(*Fault1233 - R23 Ack ID Fault*)
		Fault_Tmrs[1233].PT:= Short_Faults;
		Fault_Tmrs[1233]();
		Fault_Tmrs[1233].IN:= (GTAC_CONFIG.Option_Robot_Count>=23) AND
							MAIN.R23.Ack_ID_FLT;
		Out_To_ICxx.System_Faults[1233]:=Fault_Tmrs[1233].Q;
	(*Fault1234 - R24 Ack ID Fault*)
		Fault_Tmrs[1234].PT:= Short_Faults;
		Fault_Tmrs[1234]();
		Fault_Tmrs[1234].IN:= (GTAC_CONFIG.Option_Robot_Count>=24) AND
							MAIN.R24.Ack_ID_FLT;
		Out_To_ICxx.System_Faults[1234]:=Fault_Tmrs[1234].Q;
	(*Fault1235 - R25 Ack ID Fault*)
		Fault_Tmrs[1235].PT:= Short_Faults;
		Fault_Tmrs[1235]();
		Fault_Tmrs[1235].IN:= (GTAC_CONFIG.Option_Robot_Count>=25) AND
							MAIN.R25.Ack_ID_FLT;
		Out_To_ICxx.System_Faults[1235]:=Fault_Tmrs[1235].Q;
	(*Fault1236 - R26 Ack ID Fault*)
		Fault_Tmrs[1236].PT:= Short_Faults;
		Fault_Tmrs[1236]();
		Fault_Tmrs[1236].IN:= (GTAC_CONFIG.Option_Robot_Count>=26) AND
							MAIN.R26.Ack_ID_FLT;
		Out_To_ICxx.System_Faults[1236]:=Fault_Tmrs[1236].Q;
	(*Fault1237 - R27 Ack ID Fault*)
		Fault_Tmrs[1237].PT:= Short_Faults;
		Fault_Tmrs[1237]();
		Fault_Tmrs[1237].IN:= (GTAC_CONFIG.Option_Robot_Count>=27) AND
							MAIN.R27.Ack_ID_FLT;
		Out_To_ICxx.System_Faults[1237]:=Fault_Tmrs[1237].Q;
	(*Fault1238 - R28 Ack ID Fault*)
		Fault_Tmrs[1238].PT:= Short_Faults;
		Fault_Tmrs[1238]();
		Fault_Tmrs[1238].IN:= (GTAC_CONFIG.Option_Robot_Count>=28) AND
							MAIN.R28.Ack_ID_FLT;
		Out_To_ICxx.System_Faults[1238]:=Fault_Tmrs[1238].Q;
	(*Fault1239 - R29 Ack ID Fault*)
		Fault_Tmrs[1239].PT:= Short_Faults;
		Fault_Tmrs[1239]();
		Fault_Tmrs[1239].IN:= (GTAC_CONFIG.Option_Robot_Count>=29) AND
							MAIN.R29.Ack_ID_FLT;
		Out_To_ICxx.System_Faults[1239]:=Fault_Tmrs[1239].Q;
	(*Fault1240 - R30 Ack ID Fault*)
		Fault_Tmrs[1240].PT:= Short_Faults;
		Fault_Tmrs[1240]();
		Fault_Tmrs[1240].IN:= (GTAC_CONFIG.Option_Robot_Count>=30) AND
							MAIN.R30.Ack_ID_FLT;
		Out_To_ICxx.System_Faults[1240]:=Fault_Tmrs[1240].Q;

	(*-------------------------------------------------------------------------------- Robot Water Faults -------------------------------------------------------------------------------*)
	(*Fault1241 - R1 Water Fault*)
		Fault_Tmrs[1241].PT:= Short_Faults;
		Fault_Tmrs[1241]();
		Fault_Tmrs[1241].IN:= (GTAC_CONFIG.Option_Robot_Count>=1) AND
							MAIN.R1.WaterStand_FLT;
		Out_To_ICxx.System_Faults[1241]:=Fault_Tmrs[1241].Q;
	(*Fault1242 - R2 Water Fault*)
		Fault_Tmrs[1242].PT:= Short_Faults;
		Fault_Tmrs[1242]();
		Fault_Tmrs[1242].IN:= (GTAC_CONFIG.Option_Robot_Count>=2) AND
							MAIN.R2.WaterStand_FLT;
		Out_To_ICxx.System_Faults[1242]:=Fault_Tmrs[1242].Q;
	(*Fault1243 - R3 Water Fault*)
		Fault_Tmrs[1243].PT:= Short_Faults;
		Fault_Tmrs[1243]();
		Fault_Tmrs[1243].IN:= (GTAC_CONFIG.Option_Robot_Count>=3) AND
							MAIN.R3.WaterStand_FLT;
		Out_To_ICxx.System_Faults[1243]:=Fault_Tmrs[1243].Q;
	(*Fault1244 - R4 Water Fault*)
		Fault_Tmrs[1244].PT:= Short_Faults;
		Fault_Tmrs[1244]();
		Fault_Tmrs[1244].IN:= (GTAC_CONFIG.Option_Robot_Count>=4) AND
							MAIN.R4.WaterStand_FLT;
		Out_To_ICxx.System_Faults[1244]:=Fault_Tmrs[1244].Q;
	(*Fault1245 - R5 Water Fault*)
		Fault_Tmrs[1245].PT:= Short_Faults;
		Fault_Tmrs[1245]();
		Fault_Tmrs[1245].IN:= (GTAC_CONFIG.Option_Robot_Count>=5) AND
							MAIN.R5.WaterStand_FLT;
		Out_To_ICxx.System_Faults[1245]:=Fault_Tmrs[1245].Q;
	(*Fault1246 - R6 Water Fault*)
		Fault_Tmrs[1246].PT:= Short_Faults;
		Fault_Tmrs[1246]();
		Fault_Tmrs[1246].IN:= (GTAC_CONFIG.Option_Robot_Count>=6) AND
							MAIN.R6.WaterStand_FLT;
		Out_To_ICxx.System_Faults[1246]:=Fault_Tmrs[1246].Q;
	(*Fault1247 - R7 Water Fault*)
		Fault_Tmrs[1247].PT:= Short_Faults;
		Fault_Tmrs[1247]();
		Fault_Tmrs[1247].IN:= (GTAC_CONFIG.Option_Robot_Count>=7) AND
							MAIN.R7.WaterStand_FLT;
		Out_To_ICxx.System_Faults[1247]:=Fault_Tmrs[1247].Q;
	(*Fault1248 - R8 Water Fault*)
		Fault_Tmrs[1248].PT:= Short_Faults;
		Fault_Tmrs[1248]();
		Fault_Tmrs[1248].IN:= (GTAC_CONFIG.Option_Robot_Count>=8) AND
							MAIN.R8.WaterStand_FLT;
		Out_To_ICxx.System_Faults[1248]:=Fault_Tmrs[1248].Q;
	(*Fault1249 - R9 Water Fault*)
		Fault_Tmrs[1249].PT:= Short_Faults;
		Fault_Tmrs[1249]();
		Fault_Tmrs[1249].IN:= (GTAC_CONFIG.Option_Robot_Count>=9) AND
							MAIN.R9.WaterStand_FLT;
		Out_To_ICxx.System_Faults[1249]:=Fault_Tmrs[1249].Q;
	(*Fault1250 - R10 Water Fault*)
		Fault_Tmrs[1250].PT:= Short_Faults;
		Fault_Tmrs[1250]();
		Fault_Tmrs[1250].IN:= (GTAC_CONFIG.Option_Robot_Count>=10) AND
							MAIN.R10.WaterStand_FLT;
		Out_To_ICxx.System_Faults[1250]:=Fault_Tmrs[1250].Q;
	(*Fault1251 - R11 Water Fault*)
		Fault_Tmrs[1251].PT:= Short_Faults;
		Fault_Tmrs[1251]();
		Fault_Tmrs[1251].IN:= (GTAC_CONFIG.Option_Robot_Count>=11) AND
							MAIN.R11.WaterStand_FLT;
		Out_To_ICxx.System_Faults[1251]:=Fault_Tmrs[1251].Q;
	(*Fault1252 - R12 Water Fault*)
		Fault_Tmrs[1252].PT:= Short_Faults;
		Fault_Tmrs[1252]();
		Fault_Tmrs[1252].IN:= (GTAC_CONFIG.Option_Robot_Count>=12) AND
							MAIN.R12.WaterStand_FLT;
		Out_To_ICxx.System_Faults[1252]:=Fault_Tmrs[1252].Q;
	(*Fault1253 - R13 Water Fault*)
		Fault_Tmrs[1253].PT:= Short_Faults;
		Fault_Tmrs[1253]();
		Fault_Tmrs[1253].IN:= (GTAC_CONFIG.Option_Robot_Count>=13) AND
							MAIN.R13.WaterStand_FLT;
		Out_To_ICxx.System_Faults[1253]:=Fault_Tmrs[1253].Q;
	(*Fault1254 - R14 Water Fault*)
		Fault_Tmrs[1254].PT:= Short_Faults;
		Fault_Tmrs[1254]();
		Fault_Tmrs[1254].IN:= (GTAC_CONFIG.Option_Robot_Count>=14) AND
							MAIN.R14.WaterStand_FLT;
		Out_To_ICxx.System_Faults[1254]:=Fault_Tmrs[1254].Q;
	(*Fault1255 - R15 Water Fault*)
		Fault_Tmrs[1255].PT:= Short_Faults;
		Fault_Tmrs[1255]();
		Fault_Tmrs[1255].IN:= (GTAC_CONFIG.Option_Robot_Count>=15) AND
							MAIN.R15.WaterStand_FLT;
		Out_To_ICxx.System_Faults[1255]:=Fault_Tmrs[1255].Q;
	(*Fault1256 - R16 Water Fault*)
		Fault_Tmrs[1256].PT:= Short_Faults;
		Fault_Tmrs[1256]();
		Fault_Tmrs[1256].IN:= (GTAC_CONFIG.Option_Robot_Count>=16) AND
							MAIN.R16.WaterStand_FLT;
		Out_To_ICxx.System_Faults[1256]:=Fault_Tmrs[1256].Q;
	(*Fault1257 - R17 Water Fault*)
		Fault_Tmrs[1257].PT:= Short_Faults;
		Fault_Tmrs[1257]();
		Fault_Tmrs[1257].IN:= (GTAC_CONFIG.Option_Robot_Count>=17) AND
							MAIN.R17.WaterStand_FLT;
		Out_To_ICxx.System_Faults[1257]:=Fault_Tmrs[1257].Q;
	(*Fault1258 - R18 Water Fault*)
		Fault_Tmrs[1258].PT:= Short_Faults;
		Fault_Tmrs[1258]();
		Fault_Tmrs[1258].IN:= (GTAC_CONFIG.Option_Robot_Count>=18) AND
							MAIN.R18.WaterStand_FLT;
		Out_To_ICxx.System_Faults[1258]:=Fault_Tmrs[1258].Q;
	(*Fault1259 - R19 Water Fault*)
		Fault_Tmrs[1259].PT:= Short_Faults;
		Fault_Tmrs[1259]();
		Fault_Tmrs[1259].IN:= (GTAC_CONFIG.Option_Robot_Count>=19) AND
							MAIN.R19.WaterStand_FLT;
		Out_To_ICxx.System_Faults[1259]:=Fault_Tmrs[1259].Q;
	(*Fault1260 - R20 Water Fault*)
		Fault_Tmrs[1260].PT:= Short_Faults;
		Fault_Tmrs[1260]();
		Fault_Tmrs[1260].IN:= (GTAC_CONFIG.Option_Robot_Count>=20) AND
							MAIN.R20.WaterStand_FLT;
		Out_To_ICxx.System_Faults[1260]:=Fault_Tmrs[1260].Q;
	(*Fault1261 - R21 Water Fault*)
		Fault_Tmrs[1261].PT:= Short_Faults;
		Fault_Tmrs[1261]();
		Fault_Tmrs[1261].IN:= (GTAC_CONFIG.Option_Robot_Count>=21) AND
							MAIN.R21.WaterStand_FLT;
		Out_To_ICxx.System_Faults[1261]:=Fault_Tmrs[1261].Q;
	(*Fault1262 - R22 Water Fault*)
		Fault_Tmrs[1262].PT:= Short_Faults;
		Fault_Tmrs[1262]();
		Fault_Tmrs[1262].IN:= (GTAC_CONFIG.Option_Robot_Count>=22) AND
							MAIN.R22.WaterStand_FLT;
		Out_To_ICxx.System_Faults[1262]:=Fault_Tmrs[1262].Q;
	(*Fault1263 - R23 Water Fault*)
		Fault_Tmrs[1263].PT:= Short_Faults;
		Fault_Tmrs[1263]();
		Fault_Tmrs[1263].IN:= (GTAC_CONFIG.Option_Robot_Count>=23) AND
							MAIN.R23.WaterStand_FLT;
		Out_To_ICxx.System_Faults[1263]:=Fault_Tmrs[1263].Q;
	(*Fault1264 - R24 Water Fault*)
		Fault_Tmrs[1264].PT:= Short_Faults;
		Fault_Tmrs[1264]();
		Fault_Tmrs[1264].IN:= (GTAC_CONFIG.Option_Robot_Count>=24) AND
							MAIN.R24.WaterStand_FLT;
		Out_To_ICxx.System_Faults[1264]:=Fault_Tmrs[1264].Q;
	(*Fault1265 - R25 Water Fault*)
		Fault_Tmrs[1265].PT:= Short_Faults;
		Fault_Tmrs[1265]();
		Fault_Tmrs[1265].IN:= (GTAC_CONFIG.Option_Robot_Count>=25) AND
							MAIN.R25.WaterStand_FLT;
		Out_To_ICxx.System_Faults[1265]:=Fault_Tmrs[1265].Q;
	(*Fault1266 - R26 Water Fault*)
		Fault_Tmrs[1266].PT:= Short_Faults;
		Fault_Tmrs[1266]();
		Fault_Tmrs[1266].IN:= (GTAC_CONFIG.Option_Robot_Count>=26) AND
							MAIN.R26.WaterStand_FLT;
		Out_To_ICxx.System_Faults[1266]:=Fault_Tmrs[1266].Q;
	(*Fault1267 - R27 Water Fault*)
		Fault_Tmrs[1267].PT:= Short_Faults;
		Fault_Tmrs[1267]();
		Fault_Tmrs[1267].IN:= (GTAC_CONFIG.Option_Robot_Count>=27) AND
							MAIN.R27.WaterStand_FLT;
		Out_To_ICxx.System_Faults[1267]:=Fault_Tmrs[1267].Q;
	(*Fault1268 - R28 Water Fault*)
		Fault_Tmrs[1268].PT:= Short_Faults;
		Fault_Tmrs[1268]();
		Fault_Tmrs[1268].IN:= (GTAC_CONFIG.Option_Robot_Count>=28) AND
							MAIN.R28.WaterStand_FLT;
		Out_To_ICxx.System_Faults[1268]:=Fault_Tmrs[1268].Q;
	(*Fault1269 - R29 Water Fault*)
		Fault_Tmrs[1269].PT:= Short_Faults;
		Fault_Tmrs[1269]();
		Fault_Tmrs[1269].IN:= (GTAC_CONFIG.Option_Robot_Count>=29) AND
							MAIN.R29.WaterStand_FLT;
		Out_To_ICxx.System_Faults[1269]:=Fault_Tmrs[1269].Q;
	(*Fault1270 - R30 Water Fault*)
		Fault_Tmrs[1270].PT:= Short_Faults;
		Fault_Tmrs[1270]();
		Fault_Tmrs[1270].IN:= (GTAC_CONFIG.Option_Robot_Count>=30) AND
							MAIN.R30.WaterStand_FLT;
		Out_To_ICxx.System_Faults[1270]:=Fault_Tmrs[1270].Q;

